this is a decoder for a DCF77 signal.
the decoder decodes the DCF77 signal and checks for a valid Date_Time.
since the dcf77 signal is only secured with a simple parity the decoder waits for two consecutive valid transmissions before it sets the output signals.
given a valid reception by the receiver the decoder can take up to 3 minutes to start its clocks the first time.
after a valid signal is detected the error output goes low and dignals a valid dcf signal from the receiver.
a tp is only valid for one program cycle to allow for external rtc setting.
after a valid signal is detected two independent internal clocks are started (RTC and RTC1), the seconds  of these clocks are generated by software since the dcf signal is only valid for minutes.
rtc is always utc ( world time) and rtc1 can be set to any time zone by setting the time_zone_offset and enabling dst for automatic summertime.
a sync output signals the the rtc and rtc1 are in sync with the dcf77 signal, if the dcf77 signal is lost for more then the sync time the sync output goes low
but the rtc and rtc1 outputs keep running based on software timing until a valid dcf77 signal is received again and triggers the clock.
in addition a millisecond output gives further resolutionof the clocks.
a dst output shows if daylight saving time is enables and the weekday output shows which day of week currently is ( 1= monday ... 7= sunday).

*)

(* if tp was set it should only be active for 1 cycle *)
TP := FALSE;

(* read system time *)
t1 := DWORD_TO_TIME(T_PLC_MS());
tx := t1 - last;

IF rec XOR edge THEN
	edge := rec;
	IF NOT rec AND tx > t#1700ms AND tx < t#2000ms THEN
		(* start condition reached *)
		state := 0;
		tp := NOT error;
	ELSIF NOT rec AND tx > t#700ms AND tx < t#1000ms THEN
		(* second switch detected *)
		IF state < 58 THEN state := state +1; ELSE state := 0; END_IF;
	ELSIF rec AND tx  < t#120ms THEN
		(* bit 0 detected  *)
		bits[state] := 0;
	ELSIF rec AND tx > t#120ms AND tx < t#250ms THEN
		(* bit 1 detected *)
		bits[state] := 1;
	ELSE
		(* error condition received signal is not valid *)
		error := TRUE;
		state := 0;
	END_IF;
	last := last + tx;
	IF rec AND state = 58 THEN
		error := FALSE;

		(* decode the bits and check for possible errors *)
		IF bits[0] OR NOT (bits[17] XOR bits[18]) OR NOT bits[20] THEN error := TRUE; END_IF;
		(* decode minute *)
		MINUTE := 0;
		MINUTE.0 := bits[21];
		MINUTE.1 := bits[22];
		MINUTE.2 := bits[23];
		MINUTE.3 := bits[24];
		IF bits[25] THEN MINUTE := MINUTE + 10; END_IF;
		IF bits[26] THEN MINUTE := MINUTE + 20; END_IF;
		IF bits[27] THEN MINUTE := MINUTE + 40; END_IF;
		IF MINUTE > 59 OR (bits[21] XOR bits[22] XOR bits[23] XOR bits[24] XOR bits[25] XOR bits[26] XOR bits[27] XOR bits[28]) THEN error := TRUE; END_IF;

		(* decode hour *)
		HOUR := 0;
		HOUR.0 := bits[29];
		HOUR.1 := bits[30];
		HOUR.2 := bits[31];
		HOUR.3 := bits[32];
		IF bits[33] THEN HOUR := HOUR + 10; END_IF;
		IF bits[34] THEN HOUR := HOUR +20; END_IF;
		IF HOUR > 23 OR (bits[29] XOR bits[30] XOR bits[31] XOR bits[32] XOR bits[33] XOR bits[34] XOR bits[35]) THEN error := TRUE; END_IF;

		(* decode day of month *)
		day := 0;
		day.0 := bits[36];
		day.1 := bits[37];
		day.2 := bits[38];
		day.3 := bits[39];
		IF bits[40] THEN day := day + 10; END_IF;
		IF bits[41] THEN day := day + 20; END_IF;
		IF day > 31 THEN error := TRUE; END_IF;

		(* decode day of week *)
		wday := 0;
		wday.0 := bits[42];
		wday.1 := bits[43];
		wday.2 := bits[44];
		IF wday > 7 OR wday < 1 THEN error := TRUE; END_IF;

		(* decode month *)
		MONTH := 0;
		MONTH.0 := bits[45];
		MONTH.1 := bits[46];
		MONTH.2 := bits[47];
		MONTH.3 := bits[48];
		IF bits[49] THEN MONTH := MONTH +10; END_IF;
		IF MONTH > 12 THEN error := TRUE; END_IF;

		(* decode year *)
		YEAR := 0;
		YEAR.0 := bits[50];
		YEAR.1 := bits[51];
		YEAR.2 := bits[52];
		YEAR.3 := bits[53];
		IF bits[54] THEN YEAR := YEAR + 10; END_IF;
		IF bits[55] THEN YEAR := YEAR + 20; END_IF;
		IF bits[56] THEN YEAR := YEAR + 40; END_IF;
		IF bits[57] THEN YEAR := YEAR + 80; END_IF;

		(* check parity for bits 36 to 58 *)
		cnt := 0;
		FOR i := 36 TO 58 DO IF bits[i] THEN cnt := cnt + 1; END_IF; END_FOR;
		IF NOT EVEN(cnt) THEN error := TRUE; END_IF;

		(* time must be valid for two cycles to clear error flag *)
		IF NOT error THEN
			(* set outputs *)
			old_time := mez;
			IF YEAR >= 70 THEN YEAR := YEAR + 1900; ELSE YEAR := YEAR + 2000; END_IF;
			mez := SET_DT(YEAR,MONTH,day,HOUR,MINUTE,0);
			DS := bits[17];
			IF DS THEN
				UTC := DWORD_TO_DT(DT_TO_DWORD(mez) - 7200);
			ELSE
				UTC := DWORD_TO_DT(DT_TO_DWORD(mez) - 3600);
			END_IF;

			(* set trigger signal only if the receiver has received 2 successive minutes *)
			IF mez <> old_time + t#1m THEN error := TRUE ; END_IF;
		END_IF;
	END_IF;
END_IF;

(* this portion implements a free running clock which is triggered by the dcf77 signal *)
tz := DWORD_TO_TIME(INT_TO_DWORD(ABS(time_offset))* 3600000);

(* input sdt is copied to utc at first power up *)
IF NOT init OR SET THEN
	init := TRUE;
	utc := sdt;
	tp := TRUE;
	DS := DSI;
END_IF;

IF tp THEN
	rtc := utc;
	IF DS AND dst_en THEN
		IF time_offset < 0 THEN	rtc1 := rtc - tz + t#1h; ELSE rtc1 := rtc + tz + t#1h; END_IF;
	ELSE
		IF time_offset < 0 THEN rtc1 := rtc - tz; ELSE rtc1 := rtc + tz; END_IF;
	END_IF;
	sync := TRUE;
	last_sync := last;
	ty := last;
ELSIF rtc > DWORD_TO_DT(0) AND T1 - ty >= t#1s THEN
	rtc := rtc + t#1s;
	rtc1 := rtc1 + t#1s;
	ty := ty + t#1s;
	sync := ty - last_sync < sync_timeout AND last_sync > DWORD_TO_TIME(0);
	wday := DAY_OF_WEEK(DT_TO_DATE(rtc1));
	DS := dst_en AND DST(utc);
END_IF;
msec := TIME_TO_INT(t1 - ty);



(* decode information
bits		content
0			Bitwert immer 0
1 bis 14	reserviert für Betriebsinformationen (nicht für DCF77-Nutzer bestimmt)
15			Rufbit für Alarmierung der PTB-Mitarbeiter
			(bis Mai 2003: Bitwert = 0 falls normale Antenne in Verwendung; 1 = Backupantenne)
16			Bitwert = 1 falls ein Wechsel von MEZ nach MESZ oder umgekehrt bevorsteht; Dauer der Anzeige: 1 Stunde
17 + 18	gültige Zeit = MEZ, falls Bit 17=0 und Bit 18=1
			gültige Zeit = MESZ, falls Bit 17=1 und Bit 18=0
19			Bitwert = 1 falls innerhalb den nächsten 59 Minuten eine Schaltsekunde angeordnet ist. Beim Einfügen einer Schaltsekunde wird anstelle der 59. die 60. Sekundenmarke weggelassen und in der 58. erfolgt ausnahmsweise ein Trägerabfall.
20			Startbit für Zeitinformation (immer 1)
21 - 27		1, 2, 4, 8, 10, 20, 40 Minuten (bitweise Addition)
28			Prüfbit (gerade Parität) für die Bits 21-27
29 - 34		1, 2, 4, 8, 10, 20 Stunden (bitweise Addition)
35			Prüfbit (gerade Parität) für die Bits 29-34
36 - 41		Tagesnummer im aktuellen Monat: 1, 2, 4, 8, 10, 20 (bitweise Addition)
42 - 44		Tagesnummer in der aktuellen Woche: 1, 2, 4 (bitweise Addition)
45 - 49		Monatsnummer: 1, 2, 4, 8, 10 (bitweise Addition)
50 - 57		Jahr (zweistellig): 1, 2, 4, 8, 10, 20, 40, 80 (bitweise Addition)
58			Prüfbit (gerade Parität) füR die Bits 36-57

*)
(* revision history

hm 2.feb 2007		rev 1.1
	change wday and dst outputs when there is no dcf reception

hm	26.feb 2007		rev 1.2
	changed statements where t#1h would be substracted from DT.
	under certain conditions the compiler would crash translating this statement

hm	17. sep 2007	rev 1.3
	replaced time() with T_PLC_MS() for compatibility reasons

hm	24. oct 2007		rev 1.4
	changed dst calculation because function dst was upgraded no error in DCF77 only a change in DST

hm	12. nov 2007		rev 1.5
	changed time_offset from time to integer to allow for negative offset time zones

hm	8. dec 2007		rev 1.6
	corrected an error in time_zone calculation

hm 23. jan 2008		rev 1.7
	added sdt input which is used to initialize rtc and rtc1 during first cycle.

hm 16. mar 2008		rev 1.8
	changed output weekday to wday and dst to ds for compatibility reasons

hm	19. apr. 2008	rev 1.9
	added input dsi to allow to set daylight savings time when SDT is TRUE.
	added asynchronous SET input

hm	7. oct. 2008	rev 1.10
	changed function weekday to day_of_week

*)

END_FUNCTION_BLOCK

// POUs/Logic/gate logic/PARITY
FUNCTION PARITY : BOOL
VAR_INPUT
	in : DWORD;
END_VAR


(*
	version 1.3	18 feb 2008
	programmer 	hugo
	tested BY		hans

this function calculates the even parity of an input Dword
the output will be true if the amount of high bits are an odd number.

*)

WHILE in > 0 DO
	PARITY := PARITY XOR in.0 XOR in.1 XOR in.2 XOR in.3;
	in := SHR(in,4);
END_WHILE;

(* code before rev 1.2
WHILE in > 0 DO
	IF in.0 THEN cnt := cnt +1; END_IF;
	in := SHR(in,1);
END_WHILE;
IF (cnt MOD 2) = 1 THEN parity := TRUE; ELSE parity := FALSE; END_IF;
*)

(* revision history

rev 1.0 hm 1 sep 2006
	original version

rev 1.1 hm 10.9.2007
	changed algorithm to improve performance

rev 1.2	hm	8 dec 2007
	changed algorithm to improve performance

rev 1.3	hm	18 feb 2008
	changed algorithm to improve performance
*)

END_FUNCTION

// POUs/Engineering/control/DEAD_BAND
FUNCTION DEAD_BAND : REAL
VAR_INPUT
	X : REAL;
	L : REAL;
END_VAR


(*
version 1.2	18. jan. 2011
programmer 	hugo
tested by		oscat

DEAD_BAND ist eine lineare Übertragungsfunktion mit Totzone. Die Funktion verschiebt den positiven Teil der Kurve um +L und den negativen Teil der Kurve um -L.
DEAD_BAND = X - L wenn X > L)
DEAD_BAND = X + L wenn X < -L
DEAD_BAND = 0 wenn Abs(X) <= L

*)

IF X > L THEN
	DEAD_BAND := X - L;
ELSIF X < -L THEN
	DEAD_BAND := X + L;
ELSE
	DEAD_BAND := 0.0;
END_IF;


(* revision history
hm	2. nov. 2007	rev 1.0
	original version

hm	14. jun. 2008	rev 1.1
	improved performance

hm	18. jan. 2011	rev 1.2
	assign 0 before return
*)

END_FUNCTION

// POUs/Engineering/control/DEAD_BAND_A
FUNCTION_BLOCK DEAD_BAND_A
VAR_INPUT
	X : REAL;
	T : TIME;
	KL : REAL := 1.0;
	LM : REAL;
END_VAR
VAR_OUTPUT
	Y : REAL;
	L : REAL;
END_VAR
VAR
	tp1 : FT_PT1;
	tp2 : FT_PT1;
END_VAR


(*
version 1.1	11. mar. 2009
programmer 	hugo
tested by		oscat

DEAD_BAND ist eine lineare Übertragungsfunktion mit Totzone. Die Funktion verschiebt den positiven Teil der Kurve um -L und den negativen Teil der Kurve um +L.
DEAD_BAND = X wenn Abs(X) > L wenn Abs(X) > L
DEAD_BAND = 0 wenn Abs(X) <= L
Die Breite der Totzone wird automatisch aus dem Signalrauschen errechnet.

*)

(* filter the input signal *)
tp1(in := X, T:= T);

(* filter the HF portion to generate a stable L *)
tp2(in := ABS(tp1.out - X), T := MULTIME(T, 4.0));

(* now we determine L which is half the width of the dead band *)
L := MIN(KL * tp2.out, LM);

IF X > L THEN
	Y := X - L;
ELSIF X < -L THEN
	Y := X + L;
ELSE
	Y := 0.0;
END_IF;


(* revision history
hm	14. jun. 2008	rev 1.0
	original version

hm	11. mar. 2009	rev 1.1
	real constants updated to new systax using dot

*)

END_FUNCTION_BLOCK

// POUs/Time&Date/MULTIME
FUNCTION MULTIME : TIME
VAR_INPUT
	t : TIME;
	M : REAL;
END_VAR


(*
version 1.1	14 mar 2008
programmer 	hugo
tested by		tobias

multiplies a time by a real number and returns a time
*)

MULTIME := DWORD_TO_TIME(REAL_TO_DWORD(DWORD_TO_REAL(TIME_TO_DWORD(t))*M));

(* revision history
hm		2. oct 2006	rev 1.0
	original version

hm		14. mar 2008	rev 1.1
	rounded the result after the last digit

*)

END_FUNCTION

// POUs/Engineering/control/FT_PT1
FUNCTION_BLOCK FT_PT1
VAR_INPUT
	in : REAL;
	T : TIME;
	K : REAL := 1.0;
END_VAR
VAR_OUTPUT
	out : REAL;
END_VAR
VAR
	last : DWORD;
	tx: DWORD;
	init: BOOL;
END_VAR

(*
version 1.11	18. jan. 2011
programmer 	hugo
tested by		oscat

FT_PT1 is an low pass filter with a programmable time T and faktor K.
 
*)

(* read system time *)
tx := T_PLC_US();

(* startup initialisation *)
IF NOT init OR T = t#0s THEN
	init := TRUE;
	out := K * in;
ELSE
	out := out + (in * K - out) * DWORD_TO_REAL(Tx - last) / TIME_TO_REAL(T) * 1.0E-3;
	IF ABS(out) < 1.0E-20 THEN out := 0.0; END_IF;
END_IF;
last := tx;


(*
hm 1.1.2007	rev 1.1
	corrected error while startup value was not correct
	for very small time values real output would run out of range.

hm 3.1.2007	rev 1.2
	corrected an error for falling edge failures.
	added output faktor K.

hm 27. 2. 2007	rev 1.3
	output will be input during init for definitive startup condition.

hm	15.9.2007	rev 1.4
	changed time() to T_PLC_US() for compatibilitxy resons
	increased internal accuracy to Microseconds instead of Milliseconds

hm	23. oct 2007	rev 1.5
	added out := in to the init statements

hm	30. nov 2007	rev 1.6
	changed out to be K * in during initialization

hm	5. jan 2008	rev 1.7
	improved code for better performance

hm	16. mar. 2008	rev 1.8
	added type conversion to avoid warning under codesys 3.0

hm	14. jun. 2008	rev 1.9
	improved code

hm	11. mar. 2009	rev 1.10
	real constants updated to new systax using dot

hm	18. jan. 2011	rev 1.11
	avoid underrun of out
*)

END_FUNCTION_BLOCK

// POUs/Logic/gate logic/DEC_2
FUNCTION_BLOCK DEC_2
VAR_INPUT
	D: BOOL;
	A: BOOL;
END_VAR
VAR_OUTPUT
	Q0: BOOL;
	Q1: BOOL;
END_VAR


(*
version 1.1	3 Mar 2007
programmer 	hugo
tested by		tobias

a bit input will be decoded to the two outputs Q0 or Q1
dependent on the value of A
A=0 decodes to Q0 and A=1 decodes to Q1

*)

Q0 := D AND NOT A;
Q1 := D AND A;

(* revision history
hm 3.3.2007	rev 1.1
	rewritten in ST for better compatibility

*)

END_FUNCTION_BLOCK

// POUs/Logic/gate logic/DEC_4
FUNCTION_BLOCK DEC_4
VAR_INPUT
	D: BOOL;
	A0: BOOL;
	A1: BOOL;
END_VAR
VAR_OUTPUT
	Q0: BOOL;
	Q1: BOOL;
	Q2: BOOL;
	Q3: BOOL;
END_VAR


(*
version 1.1	3 Mar 2007
programmer 	hugo
tested by		tobias

a bit input will be decoded to one of the 4 outputs
dependent on the Adress on A0 and A1

executioin TIME on wago 750-841 = 9us
*)

Q0 := D AND NOT A0 AND NOT A1;
Q1 := D AND A0 AND NOT A1;
Q2 := D AND NOT A0 AND A1;
Q3 := D AND A0 AND A1;

(* revision history
hm 3.3.2007	rev 1.1
	rewritten in ST for better compatibility

*)

END_FUNCTION_BLOCK

// POUs/Logic/gate logic/DEC_8
FUNCTION_BLOCK DEC_8
VAR_INPUT
	D: BOOL;
	A0: BOOL;
	A1: BOOL;
	A2: BOOL;
END_VAR
VAR_OUTPUT
	Q0: BOOL;
	Q1: BOOL;
	Q2: BOOL;
	Q3: BOOL;
	Q4: BOOL;
	Q5: BOOL;
	Q6: BOOL;
	Q7: BOOL;
END_VAR
VAR
	X : INT;
END_VAR

(*
version 1.3	28. mar. 2009
programmer 	hugo
tested by		oscat

a bit input will be decoded to one of the 8 outputs
dependent on the Adress on A0, A1 and A2


*)

X.0 := A0; X.1 := A1; X.2 := A2;

Q0 := FALSE;
Q1 := FALSE;
Q2 := FALSE;
Q3 := FALSE;
Q4 := FALSE;
Q5 := FALSE;
Q6 := FALSE;
Q7 := FALSE;

CASE X OF
	0 : Q0 := D;
	1 : Q1 := D;
	2 : Q2 := D;
	3 : Q3 := D;
	4 : Q4 := D;
	5 : Q5 := D;
	6 : Q6 := D;
	7 : Q7 := D;
END_CASE;



(* revision history
hm 3. mar. 2007	rev 1.1
	rewritten in ST for better compatibility

hm	26. oct. 2008	rev 1.2
	code optimized

hm	28. mar. 2009	rev 1.3
	replaced multiple assignments
*)

END_FUNCTION_BLOCK

// POUs/String/DEC_TO_BYTE
FUNCTION DEC_TO_BYTE : BYTE
VAR_INPUT
	DEC : STRING(10);
END_VAR
VAR
	pt : POINTER TO BYTE;
	i: INT;
	X: BYTE;
	stop: INT;
END_VAR

(*
version 1.1	30. sep 2008
programmer 	hugo
tested by		oscat

DEC_TO_byte converts a decimal string into a byte.

*)

pt := ADR(dec);
stop := LEN(DEC);
FOR I := 1 TO stop DO
	(* read the first character and subtract 48 to get value in decimal 0 = 48 *)
	x := pt^;
	(* calculate the value of the digit *)
	IF X > 47 AND x < 58 THEN
		DEC_TO_BYTE := DEC_TO_BYTE * 10 + X - 48;
	END_IF;
	pt := pt + 1;
END_FOR;



(* revision histroy
hm	20. jun. 2008	rev 1.0
	original release

hm	30. sep.2008	rev 1.1
	changed length of input string from 20 to 10
	corrected an error where decoding of characters 8 and 9 would fail

*)

END_FUNCTION

// POUs/String/DEC_TO_DWORD
FUNCTION DEC_TO_DWORD : DWORD
VAR_INPUT
	DEC : STRING(20);
END_VAR
VAR
	pt : POINTER TO BYTE;
	i: INT;
	X: BYTE;
	stop: INT;
END_VAR

(*
version 1.1	30. sep. 2008
programmer 	hugo
tested by		oscat

DEC_TO_DWORD converts a decimal string into a DWORD.

*)

pt := ADR(dec);
stop := LEN(dec);
FOR I := 1 TO stop DO
	(* read the first character and subtract 48 to get value in decimal 0 = 48 *)
	x := pt^;
	(* calculate the value of the digit *)
	IF X > 47 AND x < 58 THEN
		DEC_TO_DWORD := DEC_TO_DWORD * 10 + X - 48;
	END_IF;
	pt := pt + 1;
END_FOR;



(* revision histroy
hm	20. jun. 2008	rev 1.0
	original release

hm	30. sep. 2008	rev 1.1
	corrected an error where decoding of characters 8 and 9 would fail
*)

END_FUNCTION

// POUs/String/DEC_TO_INT
FUNCTION DEC_TO_INT : INT
VAR_INPUT
	DEC : STRING(10);
END_VAR
VAR
	pt : POINTER TO BYTE;
	i: INT;
	X: BYTE;
	sign: BOOL;
	stop: INT;
END_VAR

(*
version 1.1	30. sep. 2008
programmer 	hugo
tested by	oscat

DEC_TO_INT converts a decimal string into an Integer.

*)

pt := ADR(dec);
stop := LEN(dec);
FOR I := 1 TO stop DO
	(* read the first character and subtract 48 to get value in decimal 0 = 48 *)
	x := pt^;
	(* calculate the value of the digit *)
	IF X > 47 AND x < 58 THEN
		DEC_TO_INT := DEC_TO_INT * 10 + X - 48;
	ELSIF X = 45 AND DEC_TO_INT = 0 THEN
		sign := TRUE;
	END_IF;
	pt := pt + 1;
END_FOR;
IF sign THEN DEC_TO_INT := -DEC_TO_INT; END_IF;


(* revision histroy
hm	20. jun. 2008	rev 1.0
	original release

hm	30. sep. 2008	rev 1.1
	changed length of input string from 20 to 10
	corrected an error where decoding of characters 8 and 9 would fail
*)

END_FUNCTION

// POUs/Mathematical/DEC1
FUNCTION DEC1 : INT
VAR_INPUT
	X : INT;
	N : INT;
END_VAR


(*
version 1.1	27. oct. 2008
programmer 	hugo
tested by	oscat

This is a decrement function which decrements the variable X by 1 and if 0 is reached, it begins with N-1 again.
_dec1(X,3) will generate 2,1,0,2,...

*)

IF X = 0 THEN
	DEC1 := N - 1;
ELSE
	DEC1 := X - 1;
END_IF;


(* this is a very elegant version but 50% slower
X := (X - 1 + N) MOD N;
*)


(* revision history
hm	13. oct. 2008	rev 1.0
	original version

hm	27. oct. 2008	rev 1.1
	added statement to return value for compatibility reasons

*)

END_FUNCTION

// POUs/Engineering/conversion/DEG_TO_DIR
FUNCTION DEG_TO_DIR : STRING(3)
VAR_INPUT
	DEG : INT;
	N : INT;
	L : INT;
END_VAR
VAR
	ly: INT;
END_VAR


(*
version 1.1	22. oct. 2008
programmer 	hugo
tested by		oscat

this function converts degrees in compass direction.
the function supports output in english (L=0) and german (L=1).

*)

IF L = 0 THEN ly := LANGUAGE.DEFAULT; ELSE ly := MIN(L, LANGUAGE.LMAX); END_IF;
DEG_TO_DIR := LANGUAGE.DIRS[ly, ((SHL(DEG,N-1) + 45) / 90) MOD SHL(INT#2,N)*SHR(INT#8,N)];



(*
DIR := ((SHL(DEG,N-1) + 45) / 90) MOD SHL(INT#2,N);
explanation :
DIR is calculated BY the following formula:
DIR := ((DIR + 45) / 90) MOD 4 if N = 1 digit
North = 0, East = 1 ....
DIR := ((DIR + 22,5) / 45) MOD 8 if N = 2 digit
convert to integer calculation
DIR := ((DIR*2 + 45) / 90) MOD 8
N = 0, NE = 1 ....
ther above formula replaces 2^N with shift for performance
*)



(* revision histroy
hm	11. jun. 2008	rev 1.0
	original release

hm	22. oct. 2008	rev 1.1
	changed size of string variables to 30
*)

END_FUNCTION

// POUs/String/DEL_CHARS
FUNCTION DEL_CHARS : STRING(STRING_LENGTH)
VAR_INPUT
	IN : STRING(STRING_LENGTH);
	CX : STRING(80);
END_VAR
VAR
	pos: INT := 1;
	stop: INT;
END_VAR


(*
version 1.0	18. jun. 2008
programmer 	hugo
tested by	oscat

del_chars deletes all characters from a string which are specified in CX.

*)

(* copy input string *)
DEL_CHARS := IN;
stop := LEN(in);
WHILE pos <= stop DO
	IF FIND(cx, MID(DEL_CHARS, 1, pos)) > 0 THEN
		(* wrong chracter needs to be deleted *)
		DEL_CHARS := DELETE(DEL_CHARS, 1, pos);
		stop := stop - 1;	(* the string is one character shorter now *)
	ELSE
		(* charcter not found skip to next one *)
		pos := pos + 1;
	END_IF;
END_WHILE;



(* revision history

hm		18. jun. 2008	rev 1.0		
	original version 


*)

END_FUNCTION

// POUs/Engineering/signal processing/DELAY_4
FUNCTION_BLOCK DELAY_4
VAR_INPUT
	in : REAL;
END_VAR
VAR_OUTPUT
	out1 : REAL;
	out2 : REAL;
	out3 : REAL;
	out4 : REAL;
END_VAR
VAR
	temp: REAL;
END_VAR

(*
version 1.1	19 jan 2007
programmer 	hugo
tested by		tobias

this function block delays input values by each programm cycle
after 4 cycles the in value has shifted to the out 4 and will be discarded after the next cycle
the blocks can be cascaded.

*)

out4 := out3;
out3 := out2;
out2 := out1;
out1 := temp;
temp := in;

(* revision history

hm 19.1.2007	rev 1.1
	added variable temp to add 1 delay  for q1

*)

END_FUNCTION_BLOCK

// POUs/Building/HLK/DEW_RH
FUNCTION DEW_RH : REAL
VAR_INPUT
	VC : REAL;
	T : REAL;
END_VAR

(*
version 1.2	13. mar. 2009
programmer 	hugo
tested by		tobias

this function calculates the relative humidity in air for a given temperature in °C and vapor concentration in Kg/m³..

*)

DEW_RH := LIMIT(0.0, VC / DEW_CON(1.0, T), 100.0);

(* code before rev 1.1
dew_rh := VC / dew_con(100,T) * 100;
IF dew_rh > 100 THEN dew_rh := 100; END_IF;
*)

(* revision history
hm	29. apr 2007	rev 1.0
	original version

hm	2. 12. 2007	rev 1.1
	new code for better performance

hm	13. mar. 2009	rev 1.2
	real constants updated to new systax using dot

*)

END_FUNCTION

// POUs/Building/HLK/DEW_TEMP
FUNCTION DEW_TEMP : REAL
VAR_INPUT
	RH : REAL;
	T : REAL;
END_VAR
VAR CONSTANT
	a : REAL := 7.5;
	b : REAL := 237.3;
END_VAR
VAR
	V : REAL;
END_VAR

(*
version 1.6	13. mar. 2009
programmer 	hugo
tested by		oscat

this function calculates the dew point for air given the temperature and relative humidity.
dew_temp(60,0.25) = 16.7 °C.
which means the dew point for air with 25° and 60% RH is at 16.7 °C.


*)

IF rh > 0.0 THEN
(*	old code was rewritten for better performance
	SDD := 6.1078*EXPT(10,(a*T)/(b+T));
	DD := RH/100 * SDD;
	V := LOG(DD/6.1078);
	dew_temp := b*V/(a-v);
*)
	V := LOG(RH * 0.01 * EXP10((a*T) / (b+T)));
	DEW_TEMP := b*V / (a-V);
ELSE
	DEW_TEMP:= phys.T0;
END_IF;

(* revision history

hm		2.10.2006	rev 1.0
	original version created

hm		29.4.2007	rev 1.1
	checked for rh not to be 0 because log(0) is not defined

hm		13.9.2007	rev 1.2
	code rewritten for better performance

hm	2. dec 2007	rev 1.3
	changed code for better performance

hm	8. jan 2008	rev 1.4
	further improvement in performance

hm	18. oct. 2008	rev 1.5
	using phys constants	

hm	13. mar. 2009	rev 1.6
	real constants updated to new systax using dot
	function will now return -273.15 °C for RH = 0
*)

(*
Bezeichnungen:
r = relative Luftfeuchte
T = Temperatur in °C
TK = Temperatur in Kelvin (TK = T + 273.15)
TD = Taupunkttemperatur in °C
DD = Dampfdruck in hPa
SDD = Sättigungsdampfdruck in hPa

Parameter:
a = 7.5, b = 237.3 für T >= 0
a = 7.6, b = 240.7 für T < 0 über Wasser (Taupunkt)
a = 9.5, b = 265.5 für T < 0 über Eis (Frostpunkt)

R* = 8314.3 J/(kmol*K) (universelle Gaskonstante)
mw = 18.016 kg (Molekulargewicht des Wasserdampfes)
AF = absolute Feuchte in g Wasserdampf pro m3 Luft

Formeln:

   1. SDD(T) = 6.1078 * 10^((a*T)/(b+T))
   2. DD(r,T) = r/100 * SDD(T)
   3. r(T,TD) = 100 * SDD(TD) / SDD(T)
   4. TD(r,T) = b*v/(a-v) mit v(r,T) = log10(DD(r,T)/6.1078)
   5. AF(r,TK) = 10^5 * mw/R* * DD(r,T)/TK; AF(TD,TK) = 10^5 * mw/R* * SDD(TD)/TK 

*)

END_FUNCTION

// POUs/Building/electrical/DIMM_2
FUNCTION_BLOCK DIMM_2
VAR_INPUT
	SET : BOOL;
	VAL : BYTE := 255;
	I1 : BOOL;
	I2 : BOOL;
	RST : BOOL;
END_VAR
VAR_INPUT CONSTANT
	T_DEBOUNCE : TIME := T#10ms;
	T_ON_MAX : TIME := T#0h;
	T_DIMM_START : TIME := T#1s;
	T_DIMM: TIME := T#3s;
	MIN_ON : BYTE := 50;
	MAX_ON : BYTE := 255;
	RST_OUT : BOOL := TRUE;
	SOFT_DIMM : BOOL := TRUE;
	DBL1_TOG : BOOL;
	DBL2_TOG : BOOL;
	DBL1_SET : BOOL;
	DBL2_SET : BOOL;
	DBL1_POS : BYTE;
	DBL2_POS : BYTE;
END_VAR
VAR_OUTPUT
	Q : BOOL := FALSE;
	D1 : BOOL;
	D2 : BOOL;
END_VAR
VAR_IN_OUT
	OUT : BYTE;
END_VAR
VAR
	t1, t2 : TOF;
	dc1, dc2 : CLICK_MODE;
	t3 : TON;
	dim : _RMP_B;
END_VAR

(*
version 1.0	22. mar. 2009
programmer 	hugo
tested by	tobias

this is an intelligent dimmer interface with an autoset feature using double switch inputs
a configurable debounce timer will debounce the input signals
if t_on_max is set to anything other then 0 the output will be turned off after the max on time is reached.
the times for debounce, dimming ramp, wait time before dimming and max on time are all programmable.

the dimmer has outputs Q for on and off and also out with the analog dimm value.
two additional outputs d1 and d2 decode double clicks on i1 and i2.

*)

(* debouncing for inputs i1 and i2 *)
t1(IN := I1, PT := T_DEBOUNCE);
t2(IN := I2, PT := T_DEBOUNCE);
dc1(in := t1.Q, T_LONG := T_DIMM_START);
dc2(in := t2.Q, T_LONG := T_DIMM_START);


IF RST THEN
	IF RST_OUT THEN out := 0; END_IF;
	Q := FALSE;
	D1 := FALSE;
	D2 := FALSE;
ELSIF set THEN
	OUT := VAL;
	Q := TRUE;
ELSIF dc1.SINGLE THEN
	(* single click on i1 turns the dimmer on *)
	out := LIMIT(MAX(MIN_ON,1), out, MAX_ON);
	Q := TRUE;
ELSIF dc2.SINGLE THEN
	(* single click on i2 turns the dimmer off *)
	Q := FALSE;
ELSIF dc1.TP_LONG THEN
	(* continuous on at i1 dimms up *)
	IF NOT Q THEN
		out := SEL(SOFT_DIMM, LIMIT(MAX(MIN_ON,1), out, MAX_ON), 1);
	END_IF;
	Q := TRUE;
	dim.DIR := TRUE;
ELSIF dc2.TP_LONG THEN
	(* continuous on at i2 dimms down *)
	dim.DIR := FALSE;
END_IF;

(* set the double click output *)
IF NOT DBL1_TOG THEN D1 := FALSE; END_IF;
IF dc1.DOUBLE THEN
	IF DBL1_SET THEN
		OUT := DBL1_POS;
		Q := TRUE;
	ELSE
		D1 := NOT D1;
	END_IF;
END_IF;
IF NOT DBL2_TOG THEN D2 := FALSE; END_IF;
IF dc2.DOUBLE THEN
	IF DBL2_SET THEN
		OUT := DBL2_POS;
		Q := TRUE;
	ELSE
		D2 := NOT D2;
	END_IF;
END_IF;


(* while dimming is active ramp the output out up or down *)
dim(dir := dc2.LONG, e := dc1.LONG OR dc2.LONG , TR := T_DIMM, rmp := out);

(* turn off output if a value of 0 is reached *)
IF out = 0 THEN Q := FALSE; END_IF;

(* limit the maximum runtime *)
IF t_ON_MAX > t#0s THEN
	t3(in := q, pt := T_ON_MAX);
	Q := Q XOR t3.Q;
END_IF;




(* revision history

hm 22. mar. 2009	rev 1.0
	original version

*)

END_FUNCTION_BLOCK

// POUs/Building/electrical/DIMM_I
FUNCTION_BLOCK DIMM_I
VAR_INPUT
	SET : BOOL;
	VAL : BYTE := 255;
	IN : BOOL;
	RST : BOOL;
END_VAR
VAR_INPUT CONSTANT
	T_DEBOUNCE : TIME := T#10ms;
	T_RECONFIG : TIME := T#10s;
	T_ON_MAX : TIME := T#0h;
	T_DIMM_START : TIME := T#1s;
	T_DIMM: TIME := T#3s;
	MIN_ON : BYTE := 50;
	MAX_ON : BYTE := 255;
	SOFT_DIMM : BOOL := TRUE;
	DBL_toggle : BOOL;
	RST_OUT : BOOL;
END_VAR
VAR_OUTPUT
	Q : BOOL := FALSE;
	DBL : BOOL;
END_VAR
VAR_IN_OUT
	OUT : BYTE;
END_VAR
VAR
	config : SW_RECONFIG;
	decode : CLICK_MODE;
	t3 : TON;
	dim : _RMP_B;
	dir : BOOL;
END_VAR

(*
version 2.3	26. jan. 2009
programmer 	hugo
tested by		tobias

this is an intelligent dimmer interface with an autoset feature for "in" it will automatically detect the type of switch:
low active pulses or high high active pulses are allowd for in.
a configurable debounce timer will debounce input signals
if t_on_max is set to anything other then 0 the output will be turned off after the max on time is reached.
the times for debounce, dimming ramp, wait time before dimming and max on time are all programmable.

the dimmer has outputs Q for on and off and also out with the analog dimm value.

*)

(* the input is first sent through auto reconfiguration and debouncing *)
config(IN := IN, TD := T_DEBOUNCE, TR := T_RECONFIG);
decode(in := config.Q, T_LONG := T_DIMM_START);

IF RST THEN
	IF rst_out THEN out := 0; END_IF;
	Q := FALSE;
	dir := out > 127;
ELSIF set THEN
	out := val;
	Q := TRUE;
	(* set direction to up when value < 127 otherwise set dir down dir is reversed because next action will reverse again *)
	dir := out > 127;
ELSIF decode.SINGLE THEN
	(* a single click reverses output Q *)
	Q := NOT Q;
	(* when dimmer is turned on we need to limit out to min and max limits *)
	IF Q THEN	out := LIMIT(MAX(MIN_ON,1), out, MAX_ON);	END_IF;
	(* set the appropriate direction of dimmer dir is reversed because next action will reverse again *)
	dir := out > 127;
ELSIF decode.TP_LONG THEN
	IF NOT Q THEN
		IF SOFT_DIMM THEN
			OUT := 1;
			dir := TRUE;
		ELSE
			OUT := LIMIT(MAX(MIN_ON,1), out, MAX_ON);
			DIR := out < 127;
		END_IF;
		Q := TRUE;
	ELSE
		(* reverse direction with every long click *)
		dir := NOT dir;
	END_IF;
END_IF;

(* set the double click output *)
IF NOT dbl_toggle THEN dbl := FALSE; END_IF;
IF decode.DOUBLE THEN dbl := NOT dbl; END_IF;

(* while dimming is active ramp the output out up or down *)
dim(DIR := dir, e := decode.LONG AND Q, TR := T_DIMM, rmp := out);

(* reverse direction when limits are reached *)
IF out = 0 THEN
	dir := TRUE;
ELSIF out = 255 THEN
	dir := FALSE;
END_IF;

(* limit the maximum runtime *)
IF t_ON_MAX > t#0s THEN
	t3(in := q, pt := T_ON_MAX);
	Q := Q XOR t3.Q;
END_IF;




(* revision history

hm 22.1.2007		rev 1.1
	deleted unused structure ramp

hm 2.feb 2007		rev 1.2
	changed structure to read time() at the beginning for better time consistency if a higher priorized tak interrupts dimm_i
	added statements in case structure for state 1 to allow for short 1 cycle input pulses

hm 	15.9.2007		rev 1.3
	replaced Time() with T_PLC_MS for compatibility and performance reasons

hm	30. sep. 2008	rev 1.4
	added Input VAL to supply value for set input
	added setup parameter init_val

hm	22. oct. 2008	rev 2.0
	new code and features

hm	14. nov. 2008	rev 2.1
	added soft_dimm feature

hm	16. nov. 2008	rev 2.2
	added reset out feature

hm	26. jan. 2009	rev 2.3
	dimming will also reverse at out = 0
	rst will override set
*)

END_FUNCTION_BLOCK

// POUs/Engineering/conversion/DIR_TO_DEG
FUNCTION DIR_TO_DEG : INT
VAR_INPUT
	DIR : STRING(3);
	L : INT;
END_VAR
VAR
	ly: INT;
	i : INT;
END_VAR

(*
version 1.1	22. oct. 2008
programmer 	hugo
tested by	oscat

this function converts compass directions to degrees
it will recognize up to 3 letter directions in english and german writing.

*)

IF L = 0 THEN ly := LANGUAGE.DEFAULT; ELSE ly := MIN(L, LANGUAGE.LMAX); END_IF;
FOR i := 0 TO 15 DO
	IF language.DIRS[ly, i] = DIR THEN EXIT; END_IF;
END_FOR;
DIR_TO_DEG := SHR(i * 45 + 1, 1);






(* revision histroy
hm	22. oct. 2008	rev 1.1
	original release

*)

END_FUNCTION

// POUs/Engineering/automation/DRIVER_1
FUNCTION_BLOCK DRIVER_1
VAR_INPUT CONSTANT
	Toggle_Mode : BOOL;
	Timeout : TIME;
END_VAR
VAR_INPUT
	SET : BOOL;
	IN : BOOL;
	RST : BOOL;
END_VAR
VAR_OUTPUT
	Q : BOOL;
END_VAR
VAR
	off : TON;
	edge: BOOL;
END_VAR

(*
version 1.0	2 jan 2008
programmer 	hugo
tested by		tobias

driver_1 is a multi purpose driver.
a rising edge on in sets the output high if toggle is flase. while toggle is true, a rising edge on in toggles the output Q.
if a timeout is specified the output q will be reset to false automatically after the timeout has elapsed.
a asynchronous reset and set will force the output high or low respectively.

*)

IF off.Q THEN Q := FALSE; END_IF;
IF rst THEN
	Q := FALSE;
ELSIF set THEN
	Q := TRUE;
ELSIF IN AND NOT edge THEN
	IF toggle_mode THEN q := NOT Q; ELSE q := TRUE; END_IF;
END_IF;
edge := in;
IF timeout > t#0s THEN off(in := Q, PT := Timeout); END_IF;


(* revision history
hm	2. jan 2008		rev 1.0
	original version

*)

END_FUNCTION_BLOCK

// POUs/Engineering/automation/DRIVER_4
FUNCTION_BLOCK DRIVER_4
VAR_INPUT CONSTANT
	Toggle_Mode : BOOL;
	Timeout : TIME;
END_VAR
VAR_INPUT
	SET : BOOL;
	IN0, IN1, IN2, IN3 : BOOL;
	RST : BOOL;
END_VAR
VAR_OUTPUT
	Q0, Q1, Q2, Q3 : BOOL;
END_VAR
VAR
	d0, d1, d2, d3 : DRIVER_1;
END_VAR

(*
version 1.0	2 jan 2008
programmer 	hugo
tested by		tobias

driver_4 is a 4 channel multi purpose driver.
a rising edge on in? sets the output Q? high if toggle_mode is flase. while toggle_mode is true, a rising edge on in? toggles the output Q?.
if a timeout is specified the output Q? will be reset to false automatically after the timeout has elapsed.
a asynchronous reset and set will force the output high or low respectively.
an asynchronous set will force all outputs high simultaneously

*)

D0(Set:=set, in:=in0, rst:=rst, toggle_mode:=toggle_mode, timeout:=timeout);
D1(Set:=set, in:=in1, rst:=rst, toggle_mode:=toggle_mode, timeout:=timeout);
D2(Set:=set, in:=in2, rst:=rst, toggle_mode:=toggle_mode, timeout:=timeout);
D3(Set:=set, in:=in3, rst:=rst, toggle_mode:=toggle_mode, timeout:=timeout);
Q0 := D0.Q;
Q1 := D1.Q;
Q2 := D2.Q;
Q3 := D3.Q;


(* revision history
hm	2. jan 2008		rev 1.0
	original version

*)

END_FUNCTION_BLOCK

// POUs/Engineering/automation/DRIVER_4C
FUNCTION_BLOCK DRIVER_4C
VAR_INPUT
	IN : BOOL;
	RST : BOOL;
END_VAR
VAR_INPUT CONSTANT
	Timeout : TIME;
	SX : ARRAY[1..7] OF BYTE :=[ 1,3,7,15];
END_VAR
VAR_OUTPUT
	SN : INT;
	Q0 : BOOL;
	Q1 : BOOL;
	Q2 : BOOL;
	Q3 : BOOL;
END_VAR
VAR
	off : TON;
	edge: BOOL;
END_VAR

(*
version 1.0	23. mar. 2009
programmer 	hugo
tested by	tobias

driver_4C is a multi purpose driver.
a rising edge on in switches from S0 state S1 and the next edge to state S2 and so on.
in state S0 all outputs Q are FALSE.
The stet of the Outputs in any state S? is configurable with setup variables.
The variables S1..S5 define the states, while the sequence is terminated when a state Variable S? = 0.
The lower bits 0..3 of the state vars S? are corresponding to the Outputs Q0..Q3

*)

IF RST OR off.Q THEN
	SN := 0;
ELSIF IN AND NOT edge THEN
	SN := SN + 1;
	IF SN > 7 OR SX[SN] = 0 THEN SN := 0; END_IF;
END_IF;
edge := in;
IF SN > 0 THEN
	Q0 := SX[SN].0;
	Q1 := SX[SN].1;
	Q2 := SX[SN].2;
	Q3 := SX[SN].3;
ELSE
	Q0 := FALSE;
	Q1 := FALSE;
	Q2 := FALSE;
	Q3 := FALSE;
END_IF;

(* maximaum timeout *)
IF timeout > t#0s THEN off(in := SN > 0, PT := Timeout); END_IF;


(* revision history
hm	23. mar. 2009	rev 1.0
	original version

*)

END_FUNCTION_BLOCK

// POUs/Engineering/measurements/DT_SIMU
FUNCTION_BLOCK DT_SIMU
VAR_INPUT
	START : DT;
	SPEED : REAL := 1.0;
END_VAR
VAR_OUTPUT
	DTS : DT;
END_VAR
VAR
	tc : DWORD;
	init: BOOL;
	last: DWORD;
	tx: DWORD;
	td: DWORD;
END_VAR

(*
version 1.2	8. mar. 2009
programmer 	hugo
tested by		oscat

DT_SIMU simulates a real time clock and can be adjusted to different speeds
it can also be used in simulation to simulate a real time clock.
the peed of the clock can be increased or decreased to debug timers.
with the input start a start date-time can be specified.

*)

(* read system timer *)
tx := T_PLC_MS();
tc := REAL_TO_DWORD(DWORD_TO_REAL(tx - last) * speed);

IF NOT init THEN
	init := TRUE;
	DTS := Start;
	tc := 0;
	last := tx;
ELSIF SPEED = 0.0 THEN
	DTS := DWORD_TO_DT(DT_TO_DWORD(DTS) + 1);
ELSIF tc >= 1000 THEN
	td := (tc / 1000) * 1000;
	DTS := DTS + DWORD_TO_TIME(td);
	last := last + REAL_TO_DWORD(DWORD_TO_REAL(td) / speed);
END_IF;

(* revision history
hm	11. sep. 2008	rev 1.0
	original version

hm	16. nov	2008	rev 1.1
	added type conversions for compatibility reasons

hm	8.	mar. 2009	rev 1.2
	added increment by cycle mode

*)

END_FUNCTION_BLOCK

// POUs/Time&Date/DT_TO_SDT
FUNCTION DT_TO_SDT : SDT
VAR_INPUT
	DTI : DT;
END_VAR
VAR
	tmp : DATE;
	tdt : DWORD;
END_VAR


(*
version 1.0	18. oct 2008
programmer 	hugo
tested by	oscat

converts date_time to Structured date time (SDT)

*)

tmp := DT_TO_DATE(dti);
tdt := DT_TO_DWORD(dti) - DATE_TO_DWORD(tmp);
DT_TO_SDT.YEAR := YEAR_OF_DATE(tmp);
DT_TO_SDT.MONTH := MONTH_OF_DATE(tmp);
DT_TO_SDT.DAY := DAY_OF_MONTH(tmp);
DT_TO_SDT.WEEKDAY := DAY_OF_WEEK(tmp);
DT_TO_SDT.SECOND := DWORD_TO_INT(tdt MOD 60);
DT_TO_SDT.MINUTE := DWORD_TO_INT((tdt / 60) MOD 60);
DT_TO_SDT.HOUR := DWORD_TO_INT(tdt / 3600);

(* revision history

hm 18. oct. 2008	rev 1.0
	original version

*)

END_FUNCTION

// POUs/String/DT_TO_STRF
FUNCTION DT_TO_STRF : STRING
VAR_INPUT
	DTI : DT;
	MS : INT;
	FMT : STRING;
	LANG : INT;
END_VAR
VAR CONSTANT
	FILL : STRING(1) := '0';
	BLANK : STRING(1) := ' ';
END_VAR
VAR
	ly : INT;
	dx: DATE;
	fs: STRING(10);
	td: TOD;
	tmp : INT;
	pos : INT;
	f : INT;
END_VAR

(*
version 1.1	19. oct. 2008
programmer 	hugo
tested by	oscat

DT_TO_STRINGF converts a DATETIME input to a formatted string

*)

IF LANG < 1 THEN ly := language.DEFAULT; ELSE ly := MIN(language.LMAX, LANG); END_IF;

(* decode date and time information *)
dx := DT_TO_DATE(DTI);
td := DT_TO_TOD(DTI);

(* parse the format string *)
DT_TO_STRF := FMT;
pos := FIND(DT_TO_STRF, '#');
WHILE pos > 0 DO
	(* retrieve format identifier *)
	f := CODE(DT_TO_STRF, pos + 1);
	(* generate the return string according to the format character *)
	fs := '';
	CASE f OF
		65 : (* letter A retunrs the year in 4 digits *)
			fs := INT_TO_STRING(YEAR_OF_DATE(dx));
		66 : (* letter B returns the year in exactly 2 digits *)
			fs := RIGHT(INT_TO_STRING(YEAR_OF_DATE(dx)),2);
		67 : (* letter C returns the month with 1 or 2 digits *)
			fs := INT_TO_STRING(MONTH_OF_DATE(dx));
		68 : (* letter D returns the month with exactly 2 digits *)
			fs := INT_TO_STRING(MONTH_OF_DATE(dx));
			IF LEN(fs) < 2 THEN fs := CONCAT('0', fs); END_IF;
		69 : (* letter E returns the month with 3 characters *)
			fs := MONTH_TO_STRING(MONTH_OF_DATE(dx), ly, 3);
		70 : (* letter F returns the month with all characters *)
			fs := MONTH_TO_STRING(MONTH_OF_DATE(dx), ly, 0);
		71 : (* letter G returns the day with up to 2 digits *)
			fs := INT_TO_STRING(DAY_OF_MONTH(dx));
		72 : (* letter H returns the day of the month with exactly 2 digits *)
			fs := INT_TO_STRING(DAY_OF_MONTH(dx));
			IF LEN(fs) < 2 THEN fs := CONCAT(FILL, fs); END_IF;
		73 : (* letter I returns the weekday as the number 1..7 1 = monday *)
			fs := INT_TO_STRING(DAY_OF_WEEK(dx));
		74 : (* letter J returns the weekday in 2 character writing *)
			fs := WEEKDAY_TO_STRING(DAY_OF_WEEK(dx), ly, 2);
		75 : (* letter K returns the weekday with all characters *)
			fs := WEEKDAY_TO_STRING(DAY_OF_WEEK(dx), ly, 0);
		76 : (* letter L returns AM or PM for the given DateTime *)
			IF td >= TOD#12:00 THEN fs := 'PM'; ELSE fs := 'AM'; END_IF;
		77 : (* letter M returns the hour in 1 or 2 digit form 0..24h *)
			fs := INT_TO_STRING(HOUR(td));
		78 : (* letter N returns the hour in exactly 2 digit form 0..24h *)
			fs := INT_TO_STRING(HOUR(td));
			IF LEN(fs) < 2 THEN fs := CONCAT(FILL, fs); END_IF;
		79 : (* letter O returns the hour in 1 or 2 digit form 0..12h *)
			tmp := HOUR(td) MOD 12;
			IF tmp = 0 THEN tmp := 12; END_IF;
			fs := INT_TO_STRING(tmp);
		80 : (* letter P returns the hour in exactly 2 digit form 0..12h *)
			tmp := HOUR(td) MOD 12;
			IF tmp = 0 THEN tmp := 12; END_IF;
			fs := INT_TO_STRING(tmp);
			IF LEN(fs) < 2 THEN fs := CONCAT(FILL, fs); END_IF;
		81 : (* letter Q returns the minute of the hour in 1 or two digit form *)
			fs := INT_TO_STRING(MINUTE(td));
		82 : (* letter R returns the minute of the hour in exactly two digit form *)
			fs := INT_TO_STRING(MINUTE(td));
			IF LEN(fs) < 2 THEN fs := CONCAT(FILL, fs); END_IF;
		83 : (* letter S returns the second of the minute in 1 or two digit form *)
			fs := INT_TO_STRING(REAL_TO_INT(SECOND(td)));
		84 : (* letter T returns the second of the minute in exactly two digit form *)
			fs := INT_TO_STRING(REAL_TO_INT(SECOND(td)));
			IF LEN(fs) < 2 THEN fs := CONCAT(FILL, fs); END_IF;
		85 : (* letter U returns the milliseconds in 1 to 3 digits *)
			fs := INT_TO_STRING(MS);
		86 : (* letter V returns the milliseconds in exactly 3 digit form *)
			fs := INT_TO_STRING(MS);
			fs := CONCAT('00',fs);
			fs := RIGHT(fs, 3);
		87 : (* letter W returns the day of the month with exactly 2 digits first digit is filled with blank if necessary *)
			fs := INT_TO_STRING(DAY_OF_MONTH(dx));
			IF LEN(fs) < 2 THEN fs := CONCAT(BLANK, fs); END_IF;
		88 : (* letter X returns the month with exactly 2 digits first digit is filled with blank if necessary *)
			fs := INT_TO_STRING(MONTH_OF_DATE(dx));
			IF LEN(fs) < 2 THEN fs := CONCAT(BLANK, fs); END_IF;
		END_CASE;
	DT_TO_STRF := REPLACE(DT_TO_STRF, fs, 2, pos);
	pos := FIND(DT_TO_STRF, '#');
END_WHILE;


(* revision history
hm	7. oct. 2008	rev 1.0
	original version

hm	19. oct. 2008	rev 1.1
	changed language setup constants
*)

END_FUNCTION

// POUs/String/MONTH_TO_STRING
FUNCTION MONTH_TO_STRING : STRING(10)
VAR_INPUT
	MTH : INT;
	LANG : INT;
	LX : INT;
END_VAR
VAR
	ly : INT;
END_VAR

(*
version 1.1	19. oct. 2008
programmer 	hugo
tested by	oscat

MONTH_TO_STRING converts an Integer 1..12 into a String with the Names of the corresponding Month.
the decoding is according to the language setup in global vars

*)

IF LANG = 0 THEN Ly := LANGUAGE.DEFAULT; ELSE ly := MIN(LANG, language.LMAX); END_IF;
IF MTH < 1 OR MTH > 12 THEN
	RETURN;
ELSIF LX = 0 THEN
	MONTH_TO_STRING := language.MONTHS[ly, MTH];
ELSIF Lx = 3 THEN
	MONTH_TO_STRING := language.MONTHS3[ly, MTH];
END_IF;


(* revisison history

hm	21. sep. 2008	rev 1.0
	original version

hm	19. oct. 2008	rev 1.1
	changed language setup constants
*)

END_FUNCTION

// POUs/String/WEEKDAY_TO_STRING
FUNCTION WEEKDAY_TO_STRING : STRING(10)
VAR_INPUT
	WDAY : INT;
	LANG : INT;
	LX : INT;
END_VAR
VAR
	ly : INT;
END_VAR

(*
version 1.1	19. oct. 2008
programmer 	hugo
tested by	oscat

WEEKDAY_TO_STRING converts an Integer 1..7 into a String with the Names of the corresponding weekday.
the decoding is according to the language setup in global vars

*)

IF LANG = 0 THEN ly := LANGUAGE.DEFAULT; ELSE ly := MIN(LANG, LANGUAGE.LMAX); END_IF;
IF wday < 1 OR wday > 7 THEN
	RETURN;
ELSIF LX = 0 THEN
	WEEKDAY_TO_STRING := language.WEEKDAYS[ly, WDAY];
ELSIF Lx = 2 THEN
	WEEKDAY_TO_STRING := language.WEEKDAYS2[ly, WDAY];
END_IF;


(* revisison history

hm	21. sep. 2008	rev 1.0
	original version

hm	19. oct. 2008	rev 1.1
	changed language setup constants
*)

END_FUNCTION

// POUs/Time&Date/DT2_TO_SDT
FUNCTION DT2_TO_SDT : SDT
VAR_INPUT
	DI : DATE;
	TI : TOD;
END_VAR


(*
version 1.0	18. oct 2008
programmer 	hugo
tested by	oscat

converts date and time of day to Structured date time (SDT)

*)

DT2_TO_SDT.YEAR := YEAR_OF_DATE(di);
DT2_TO_SDT.MONTH := MONTH_OF_DATE(di);
DT2_TO_SDT.DAY := DAY_OF_MONTH(di);
DT2_TO_SDT.WEEKDAY := DAY_OF_WEEK(di);
DT2_TO_SDT.MS := DWORD_TO_INT(TOD_TO_DWORD(ti) MOD 1000);
DT2_TO_SDT.SECOND := DWORD_TO_INT((TOD_TO_DWORD(ti) / 1000) MOD 60);
DT2_TO_SDT.MINUTE := DWORD_TO_INT((TOD_TO_DWORD(ti) / 60000) MOD 60);
DT2_TO_SDT.HOUR := DWORD_TO_INT(TOD_TO_DWORD(ti) / 3600000);

(* revision history

hm 18. oct. 2008	rev 1.0
	original version

*)

END_FUNCTION

// POUs/Logic/gate logic/DW_TO_REAL
FUNCTION DW_TO_REAL : REAL
VAR_INPUT
	X : DWORD;
END_VAR
VAR
	pt : POINTER TO REAL;
END_VAR

(*
version 1.0	18. apr. 2008
programmer 	hugo
tested by		tobias

this function converts a DWORD to REAL in a bitwise manner.
*)

pt := ADR(X);
DW_TO_REAL := pt^;

(* revision history
hm	18. apr. 2008
	original version

*)

END_FUNCTION

// POUs/Logic/gate logic/DWORD_OF_BYTE
FUNCTION DWORD_OF_BYTE : DWORD
VAR_INPUT
	B3 : BYTE;
	B2 : BYTE;
	B1 : BYTE;
	B0 : BYTE;
END_VAR


(*
version 1.3	18. jul. 2009
programmer 	hugo
tested by		tobias

this function creates a Dword from 4 individual bytes

*)

DWORD_OF_BYTE := SHL(SHL(SHL(BYTE_TO_DWORD(B3),8) OR BYTE_TO_DWORD(B2),8) OR BYTE_TO_DWORD(B1),8) OR BYTE_TO_DWORD(B0);


(* revision history
hm	24. jan 2007	rev 1.0
	original version

hm 2. jan 2008	rev 1.1
	inproved performance

hm	23. apr. 2008	rev 1.2
	reverse order of inputs to be more logical

hm	18. jul. 2009	rev 1.3
	added type conversions for compatibility reasons
*)

END_FUNCTION

// POUs/Logic/gate logic/DWORD_OF_WORD
FUNCTION DWORD_OF_WORD : DWORD
VAR_INPUT
	W1 : WORD;
	W0 : WORD;
END_VAR


(*
version 1.0	18. jul. 2009
programmer 	hugo
tested by		tobias

this function creates a Dword from 2 individual Words

*)

DWORD_OF_WORD := SHL(WORD_TO_DWORD(W1),16) OR WORD_TO_DWORD(W0);


(* revision history

hm	18. jul. 2009	rev 1.0
	original version

*)

END_FUNCTION

// POUs/String/DWORD_TO_STRB
FUNCTION DWORD_TO_STRB : STRING(32)
VAR_INPUT
	IN : DWORD;
END_VAR
VAR
	pt : POINTER TO BYTE;
	i: INT;
END_VAR

(*
version 1.3	20. jun. 2008
programmer 	hugo
tested by	oscat

DWORD_TO_STRINGB converts a DWORD to a String of Bits represented by '0' and '1' s.
The lowest order bit will be on the right and the high order bit on the left.

*)

(* pointer für die ausgabe ermitteln *)
pt := ADR(DWORD_TO_STRB);
(* die 8 ausgabecharacter ermitteln und schreiben *)
FOR i := 1 TO 32 DO
	pt^:= BOOL_TO_BYTE(in.31) + 48;
	in := SHL(in,1);
	pt := pt + 1;
END_FOR;

(* der ausgabestring muss nochg mit 0 abgeschlossen werden *)
pt^ := 0;

(* revision history
hm		9.6.2007	rev 1.0		
	original version

hm		15.dec 2007	rev 1.1
	changed code for better performance

hm	29. mar. 2008	rev 1.2
	changed STRING to STRING(32)

hm	20. jun. 2008	rev 1.3
	performance improvement

*)

END_FUNCTION

// POUs/String/DWORD_TO_STRF
FUNCTION DWORD_TO_STRF : STRING(20)
VAR_INPUT
	IN : DWORD;
	N : INT;
END_VAR


(*
version 1.0	26 jan 2007
programmer 	hugo
tested by		tobias

dword_to_strF converts a DWORD, BYTE or Word to a fixed length String.
the string will be filled with leading zeroes to achieve the fixed length, or if too long, the lowest digits will be used.
the maximum allowed length is 20 mdigits.

for example:	dword_to_strf(123,4) = '0123' 
				dword_to_strf(123,2) = '23'
*)

(* limit N to max 20 characters *)
(* convert dword to string first and cut to length N *)
DWORD_TO_STRF := FIX(DWORD_TO_STRING(in),LIMIT(0,N,20),48,1);


(* revision history
hm	26. jan.2007	rev 1.0		
	original version

hm	29. mar. 2008	rev 1.1
	changed STRING to STRING(20)
	limit the output string to max 20 digits
*)

END_FUNCTION

// POUs/String/FIX
FUNCTION FIX : STRING(STRING_LENGTH)
VAR_INPUT
	str : STRING(STRING_LENGTH);
	L : INT;
	C : BYTE;
	M : INT;
END_VAR
VAR
	N : INT;
	SX: STRING(STRING_LENGTH);
END_VAR

(*
version 1.0	29. mar. 2008
programmer 	hugo
tested by	tobias

the function fix truncates a string at length L 
or if the string is shorter then L it will be filled with ending Spaces till its length = N.

*)

(* make sure L does not exceed the limits of a string *)
N := LIMIT(0,L,STRING_LENGTH) - LEN(str);
IF N <= 0 THEN
	(* truncate the string at length N *)
	IF M = 1 THEN
		FIX := RIGHT(str,L);
	ELSE
		FIX := LEFT(str,L);
	END_IF;
ELSIF M = 1 THEN
	(* connect fill characters at the beginning *)
	sx := FILL(C,N);
	FIX := CONCAT(sx,str);
ELSIF M = 2 THEN
	(* center str beween fill characters *)
	(* for an uneven number of fill characters, there is one more at the end *)
	sx := FILL(C,SHR(N+1,1));
	FIX := CONCAT(str,sx);
	SX := LEFT(sx,SHR(N,1));
	FIX := CONCAT(sx,FIX);
ELSE
	(* connect fill characters at the end *)
	SX := FILL(C,N);
	FIX := CONCAT(str,SX);
END_IF;


(* revision histroy
hm	29. mar. 2008	rev 1.0
	original release

*)

END_FUNCTION

// POUs/String/DWORD_TO_STRH
FUNCTION DWORD_TO_STRH : STRING(8)
VAR_INPUT
	IN : DWORD;
END_VAR
VAR
	i : INT;
	temp : BYTE;
	pt : POINTER TO BYTE;
END_VAR

(*
version 1.3	29. mar. 2008
programmer 	hugo
tested by	tobias

DWORD_TO_STRINGH converts a DWORD to a String of Hexadecimal represented by '0' .. '9' and 'A' .. 'F'.
The lowest order Character will be on the right and the high order Character on the left.

*)

(* read output adress to pointer *)
pt := ADR(DWORD_TO_STRH) + 8;
(* wirte the closing byte for the string *)
pt^:= 0;

(* write the 8 hex characters backwards *)
FOR i := 1 TO 8 DO;
	(* decrement the pointer *)
	pt := pt - 1;
	(* read the lowest order hex value *)
	temp := DWORD_TO_BYTE(in AND 16#0000000F);
	(* convert value to hex character *)
	IF temp <= 9 THEN temp := temp + 48; ELSE temp := temp + 55; END_IF;
	(* write character to output string *)
	PT^ := temp;
	(* shift in for nect hex character *)
	in := SHR(in,4);
END_FOR;


(* code beofre rev 1.2
FOR i := 1 TO 8 DO
	X := DWORD_TO_BYTE(in AND 2#1111);
	IF X <= 9 THEN X := X + 48; ELSE X := X + 55; END_IF;
	Cx := CHR(X);
	temp := CONCAT(Cx, temp);
	in := SHR(in,4);
END_FOR;
DWORD_TO_STRH := temp;
*)


(* revision history
hm	9. jun. 2007	rev 1.0		
	original version 

hm	11. sep. 2007	rev 1.1
	changed coding for compatibility with twincat, concat cannot support a function as an argument.

hm	15. dec. 2007	rev 1.2
	changed code for better performance

hm	29. mar. 2008	rev 1.3
	changed STRING to STRING(8)

*)

END_FUNCTION

// POUs/Mathematical/Geometry/ELLIPSE_A
FUNCTION ELLIPSE_A : REAL
VAR_INPUT
	R1 : REAL;
	R2 : REAL;
END_VAR


(*
version 1.1	18. oct. 2008
programmer 	hugo
tested by	oscat

ellipse_A calculates the Area of an ellipe based on the two radians R1 and R2


*)

ELLIPSE_A := math.PI * R1 * R2;

(* revision histroy
hm	16. oct 2007	rev 1.0
	original version

hm	18. oct. 2008	rev 1.1
	using math constants
*)

END_FUNCTION

// POUs/Mathematical/Geometry/ELLIPSE_C
FUNCTION ELLIPSE_C : REAL
VAR_INPUT
	R1 : REAL;
	R2 : REAL;
END_VAR


(*
version 1.2	10. mar. 2009
programmer 	hugo
tested by		oscat

ellipse_C calculates the circumference of an ellipe based on the two radians R1 and R2

*)

ELLIPSE_C := math.PI * (3.0 * (R1+R2) - SQRT((3.0 * r1 + R2) * (3.0 * r2 + r1)));

(* revision histroy
hm	16. oct 2007	rev 1.0
	original version

hm	18. oct. 2008	rev 1.1
	using math constants

hm	10. mar. 2009	rev 1.2
	changed syntax of real constants to 0.0

*)

END_FUNCTION

// POUs/Engineering/conversion/ENERGY
FUNCTION_BLOCK ENERGY
VAR_INPUT
	J : REAL;
	C : REAL;
	Wh : REAL;
END_VAR
VAR_OUTPUT
	YJ : REAL;
	YC : REAL;
	YWh : REAL;
END_VAR


(*
version 1.2	16. jan. 2010
programmer 	hugo
tested by		oscat

this function converts different energy units
any unused input can simply be left open.
different inputs connected at the same time will be added up.
*)

YJ := J + Wh * 3600.0 + C * 4.1868;
YC := YJ * 0.238845896627496;
YWh := YJ * 2.7777777778E-004;

(*
Arbeit, Energie, Joule* J 1 J = 1 N · m = 1 W · s = (1/3,6) E6 kW · h = 1 kg · m2/s2
Wärmemenge Kilowattstunde kW · h 1 kW · h = 3,6 MJ = 860 kcal
Elektronvolt eV 1 eV = 160,218 92 E21 J
Erg erg 1 erg = 1E7 J
Kalorie calorie 1 calalorie = 4,1868 J = 1,163 E3 W · h
Therm therm 1 therm = 105,50 · 106 J
*)

(* revision history

hm	27. mar. 2007	rev 1.0
	original version

hm	11. mar. 2009	rev 1.1
	improved code

hm 16. jan 2010	rev 1.2
	avoid the string cal in comments for codesys import bug


*)

END_FUNCTION_BLOCK

// POUs/Mathematical/ERF
FUNCTION ERF : REAL
VAR_INPUT
	X : REAL;
END_VAR
VAR
	x2 : REAL;
	ax2 : REAL;
END_VAR


(*
version 1.3	10. mar. 2009
programmer 	hugo
tested by		tobias

this function calculates the erf (error) function.

*)

x2 := X*X;
ax2 := 0.147 * x2 + 1.0;
ERF := SQRT(1.0 - EXP(-X2 * ((0.27323954473516 + aX2)/(ax2)))) * SGN(x);




(* revision history
hm	7. apr. 2008	rev 1.0
	original version

hm	30. jun. 2008	rev 1.1
	added type conversions to avoid warnings under codesys 3.0

hm	25. oct. 2008	rev 1.2
	new code using new algorithm

hm	10. mar. 2009	rev 1.3
	real constants updated to new systax using dot
*)

END_FUNCTION

// POUs/Mathematical/ERFC
FUNCTION ERFC : REAL
VAR_INPUT
	X : REAL;
END_VAR


(*
version 1.1	10. mar. 2009
programmer 	hugo
tested by		tobias

this function calculates the inverse erf (error) function.

*)

ERFC := 1.0 - ERF(X);

(* revision history
hm	7. apr. 2008	rev 1.0
	original version

hm	10. mar. 2009	rev 1.1
	real constants updated to new systax using dot

*)

END_FUNCTION

// POUs/Other/ESR_COLLECT
FUNCTION_BLOCK ESR_COLLECT
VAR_INPUT
	ESR_0, ESR_1, ESR_2, ESR_3, ESR_4, ESR_5, ESR_6, ESR_7 : ARRAY [0..3] OF esr_data;
	rst : BOOL;
END_VAR
VAR_IN_OUT
	pos : INT;
END_VAR
VAR_OUTPUT
	ESR_OUT : ARRAY[0..31] OF esr_data;
END_VAR
VAR CONSTANT
	max_in : INT := 3; (* max limit of input array *)
	max_out : INT := 32; (* number of elements in array *)
END_VAR
VAR
	cnt : INT := -1;
END_VAR

(*
version 1.4	1. dec. 2009
programmer 	hugo
tested by		tobias

ESR_collect collects esr data from up to 8 esr_mon modules and stroes them in an output array.
the output pos will display the position of the last element in the array. if the array is empty, pos = -1
when to buffer is read by followon modules. pos has to be reset to -1
if the array will be full, the buffer will be refilled starting at position 0.

*)

IF rst OR cnt < 0 THEN
	pos := -1;
ELSE
	FOR cnt := 0 TO max_in DO
	IF esr_0[cnt].typ > 0 THEN pos := INC1(pos, max_out); esr_out[pos] := esr_0[cnt]; END_IF;
	IF esr_1[cnt].typ > 0 THEN pos := INC1(pos, max_out); esr_out[pos] := esr_1[cnt]; END_IF;
	IF esr_2[cnt].typ > 0 THEN pos := INC1(pos, max_out); esr_out[pos] := esr_2[cnt]; END_IF;
	IF esr_3[cnt].typ > 0 THEN pos := INC1(pos, max_out); esr_out[pos] := esr_3[cnt]; END_IF;
	IF esr_4[cnt].typ > 0 THEN pos := INC1(pos, max_out); esr_out[pos] := esr_4[cnt]; END_IF;
	IF esr_5[cnt].typ > 0 THEN pos := INC1(pos, max_out); esr_out[pos] := esr_5[cnt]; END_IF;
	IF esr_6[cnt].typ > 0 THEN pos := INC1(pos, max_out); esr_out[pos] := esr_6[cnt]; END_IF;
	IF esr_7[cnt].typ > 0 THEN pos := INC1(pos, max_out); esr_out[pos] := esr_7[cnt]; END_IF;
   END_FOR;
END_IF;


(* revision history
hm	26.jan 2007	rev 1.0
	original version

hm	8. dec 2007	rev 1.1
	added reset input

ks	27. oct. 2008	rev 1.2
	optimized code for performance

ks	12. nov. 2009	rev 1.3
	output pos was not pointing to last value	

hm	1. dec. 2009	rev 1.4
	changed pos to be I/O
	reduced output array size to 32 elements
*)

END_FUNCTION_BLOCK

// POUs/Other/ESR_MON_B8
FUNCTION_BLOCK ESR_MON_B8
VAR_INPUT
	s0, s1, s2, s3, s4, s5, s6, s7 : BOOL;
	DT_in : DT;
END_VAR
VAR_INPUT CONSTANT
	a0, a1, a2, a3, a4, a5, a6, a7 : STRING(10);
END_VAR
VAR_OUTPUT
	ESR_Flag : BOOL;
END_VAR
VAR_IN_OUT
	ESR_Out: ARRAY [0..3] OF esr_data;
END_VAR
VAR
	x0, x1, x2, x3, x4, x5, x6, x7 : BOOL;
	tx: TIME;
	cnt : INT;
END_VAR

(*
version 1.3	1. dec. 2009
programmer 	hugo
tested by		tobias

ESR_mon_B8 monitores up to 8 binary inputs and reports changes with time stamd and adress label.
the module checks 8 inputs for a change and reports all changes with time and adress stamp to the output.
4 events maximum can be collected at once within the same cycle

*)

(* read system timer *)
tx := DWORD_TO_TIME(T_PLC_MS());

ESR_Flag := FALSE;
esr_out[3].typ := 0;
esr_out[2].typ := 0;
esr_out[1].typ := 0;
esr_out[0].typ := 0;
cnt := 0;


(* check if inputs have chaged and fill buffer *)
IF s0 <> X0 THEN
	esr_out[cnt].typ := 10 + BOOL_TO_BYTE(s0);
	esr_out[cnt].adress := a0;
	esr_out[cnt].DS := DT_in;
	esr_out[cnt].TS := TX;
	X0 := S0;
	cnt := cnt + 1;
	esr_flag := TRUE;
END_IF;
IF s1 <> X1 THEN
	esr_out[cnt].typ := 10 + BOOL_TO_BYTE(s1);
	esr_out[cnt].adress := a1;
	esr_out[cnt].DS := DT_in;
	esr_out[cnt].TS := TX;
	X1 := S1;
	cnt := cnt + 1;
	esr_flag := TRUE;
END_IF;
IF s2 <> X2 THEN
	esr_out[cnt].typ := 10 + BOOL_TO_BYTE(s2);
	esr_out[cnt].adress := a2;
	esr_out[cnt].DS := DT_in;
	esr_out[cnt].TS := TX;
	X2 := S2;
	cnt := cnt + 1;
	esr_flag := TRUE;
END_IF;
IF s3 <> X3 THEN
	esr_out[cnt].typ := 10 + BOOL_TO_BYTE(s3);
	esr_out[cnt].adress := a3;
	esr_out[cnt].DS := DT_in;
	esr_out[cnt].TS := TX;
	X3 := S3;
	cnt := cnt + 1;
	esr_flag := TRUE;
END_IF;
IF s4 <> X4 AND cnt < 4 THEN
	esr_out[cnt].typ := 10 + BOOL_TO_BYTE(s4);
	esr_out[cnt].adress := a4;
	esr_out[cnt].DS := DT_in;
	esr_out[cnt].TS := TX;
	X4 := S4;
	cnt := cnt + 1;
	esr_flag := TRUE;
END_IF;
IF s5 <> X5  AND cnt < 4 THEN
	esr_out[cnt].typ := 10 + BOOL_TO_BYTE(s5);
	esr_out[cnt].adress := a5;
	esr_out[cnt].DS := DT_in;
	esr_out[cnt].TS := TX;
	X5 := S5;
	cnt := cnt + 1;
	esr_flag := TRUE;
END_IF;
IF s6 <> X6  AND cnt < 4 THEN
	esr_out[cnt].typ := 10 + BOOL_TO_BYTE(s6);
	esr_out[cnt].adress := a6;
	esr_out[cnt].DS := DT_in;
	esr_out[cnt].TS := TX;
	X6 := S6;
	cnt := cnt + 1;
	esr_flag := TRUE;
END_IF;
IF s7 <> X7  AND cnt < 4 THEN
	esr_out[cnt].typ := 10 + BOOL_TO_BYTE(s7);
	esr_out[cnt].adress := a7;
	esr_out[cnt].DS := DT_in;
	esr_out[cnt].TS := TX;
	X7 := S7;
	cnt := cnt + 1;
	esr_flag := TRUE;
END_IF;

(* revision history
hm	26. jan 2007	rev 1.0
	original version

hm	17. sep 2007	rev 1.1
	replaced time() with T_PLC_MS() for compatibility reasons

hm	22. oct. 2008	rev 1.2
	optimized code

hm	1.dec. 2009	rev 1.3
	changed esr_out to be I/O

*)

END_FUNCTION_BLOCK

// POUs/Other/ESR_MON_R4
FUNCTION_BLOCK ESR_MON_R4
VAR_INPUT
	R0, R1, R2, R3 : REAL;
	DT_in : DT;
END_VAR
VAR_INPUT CONSTANT
	a0, a1, a2, a3 : STRING(10);
	s0, s1, s2, s3 : REAL;
END_VAR
VAR_OUTPUT
	ESR_Flag : BOOL;
END_VAR
VAR_IN_OUT
	ESR_Out: ARRAY [0..3] OF esr_data;
END_VAR
VAR
	p0, p1, p2, p3 : POINTER TO DWORD;
	x0, x1, x2, x3 : REAL;
	tx: TIME;
	cnt : INT;
END_VAR

(*
version 1.4	1. dec. 2009
programmer 	hugo
tested by		tobias

ESR_mon_R4 monitores up to 4 Real inputs and reports changes with time stamd and adress label.
the module checks 4 inputs for a change of more than the specified sensitivity S and reports all changes with time and adress stamp to the output.

*)

(* read system timer *)
tx := DWORD_TO_TIME(T_PLC_MS());
P0 := ADR(R0);
P1 := ADR(R1);
P2 := ADR(R2);
P3 := ADR(R3);

ESR_Flag := FALSE;
esr_out[3].typ := 0;
esr_out[2].typ := 0;
esr_out[1].typ := 0;
esr_out[0].typ := 0;
cnt := 0;

(* check if inputs have chaged and fill buffer *)
IF DIFFER(R0,  X0, S0) THEN
	esr_out[cnt].typ := 20;
	esr_out[cnt].adress := a0;
	esr_out[cnt].DS := DT_in;
	esr_out[cnt].TS := TX;
	esr_out[cnt].data[0] := Byte_of_Dword(P0^,0);
	esr_out[cnt].data[1] := Byte_of_Dword(P0^,1);
	esr_out[cnt].data[2] := Byte_of_Dword(P0^,2);
	esr_out[cnt].data[3] := Byte_of_Dword(P0^,3);
	X0 := R0;
	cnt := cnt + 1;
	esr_flag := TRUE;
END_IF;
IF differ(R1,  X1, S1) THEN
	esr_out[cnt].typ := 20;
	esr_out[cnt].adress := a1;
	esr_out[cnt].DS := DT_in;
	esr_out[cnt].TS := TX;
	esr_out[cnt].data[0] := Byte_of_Dword(P1^,0);
	esr_out[cnt].data[1] := Byte_of_Dword(P1^,1);
	esr_out[cnt].data[2] := Byte_of_Dword(P1^,2);
	esr_out[cnt].data[3] := Byte_of_Dword(P1^,3);
	X1 := R1;
	cnt := cnt + 1;
	esr_flag := TRUE;
END_IF;
IF differ(R2,  X2, S2) THEN
	esr_out[cnt].typ := 20;
	esr_out[cnt].adress := a2;
	esr_out[cnt].DS := DT_in;
	esr_out[cnt].TS := TX;
	esr_out[cnt].data[0] := Byte_of_Dword(P2^,0);
	esr_out[cnt].data[1] := Byte_of_Dword(P2^,1);
	esr_out[cnt].data[2] := Byte_of_Dword(P2^,2);
	esr_out[cnt].data[3] := Byte_of_Dword(P2^,3);
	X2 := R2;
	cnt := cnt + 1;
	esr_flag := TRUE;
END_IF;
IF DIFFER(R3,  X3, S3) THEN
	esr_out[cnt].typ := 20;
	esr_out[cnt].adress := a3;
	esr_out[cnt].DS := DT_in;
	esr_out[cnt].TS := TX;
	esr_out[cnt].data[0] := Byte_of_Dword(P3^,0);
	esr_out[cnt].data[1] := Byte_of_Dword(P3^,1);
	esr_out[cnt].data[2] := Byte_of_Dword(P3^,2);
	esr_out[cnt].data[3] := Byte_of_Dword(P3^,3);
	X3 := R3;
	cnt := cnt + 1;
	esr_flag := TRUE;
END_IF;


(* revision history
hm	26. jan 2007	rev 1.0
	original version

hm	17. sep. 2007		rev 1.1
	replaced time() with T_PLC_MS() for compatibility reasons

hm	8. dec. 2007		rev 1.2
	corrected an error while esr typ would not be set

hm	16. mar. 2008		rev 1.3
	deleted wrong conversion real_to_dword

hm	1. dec 2009		rev 1.4
	changed esr_out to be I/O

*)

END_FUNCTION_BLOCK

// POUs/Other/ESR_MON_X8
FUNCTION_BLOCK ESR_MON_X8
VAR_INPUT
	s0, s1, s2, s3, s4, s5, s6, s7 : BYTE;
	DT_in : DT;
	Mode : BYTE := 3;
END_VAR
VAR_INPUT CONSTANT
	a0, a1, a2, a3, a4, a5, a6, a7 : STRING(10);
END_VAR
VAR_OUTPUT
	ESR_Flag : BOOL;
END_VAR
VAR_IN_OUT
	ESR_Out: ARRAY [0..3] OF esr_data;
END_VAR
VAR
	x0, x1, x2, x3, x4, x5, x6, x7 : BYTE;
	tx: TIME;
	cnt : INT;
END_VAR

(*
version 1.2	1. dec. 2009
programmer 	hugo
tested by		tobias

ESR_MON_X8 is a status and error collector.
the module checks 8 status inputs for a change and reports up to 4 input changes with time and adress stamp to the output.
the mode can be 
1 for error only
2 for error and status
3 for error, status and debug
the adress label of the 8 inputs can be configured individually.
*)

(* read system timer *)
tx := DWORD_TO_TIME(T_PLC_MS());

ESR_Flag := FALSE;
esr_out[3].typ := 0;
esr_out[2].typ := 0;
esr_out[1].typ := 0;
esr_out[0].typ := 0;
cnt := 0;


(* check if inputs have chaged and fill buffer *)
IF s0 <> X0 AND ((s0 < 100) OR (S0 > 99 AND S0 < 200 AND mode >= 2) OR (S0 > 199 AND mode = 3)) THEN
	esr_out[cnt] := status_to_ESR(s0, a0, DT_in, TX);
	X0 := S0;
	cnt := cnt + 1;
	esr_flag := TRUE;
END_IF;
IF s1 <> X1 AND ((s1 < 100) OR (S1 > 99 AND S1 < 200 AND mode >= 2) OR (S1 > 199 AND mode = 3)) THEN
	esr_out[cnt] := status_to_ESR(s1, a1, DT_in, TX);
	X1 := S1;
	cnt := cnt + 1;
	esr_flag := TRUE;
END_IF;
IF s2 <> X2 AND ((s2 < 100) OR (S2 > 99 AND S2 < 200 AND mode >= 2) OR (S2 > 199 AND mode = 3)) THEN
	esr_out[cnt] := status_to_ESR(s2, a2, DT_in, TX);
	X2 := S2;
	cnt := cnt + 1;
	esr_flag := TRUE;
END_IF;
IF s3 <> X3 AND ((s3 < 100) OR (S3 > 99 AND S3 < 200 AND mode >= 2) OR (S3 > 199 AND mode = 3)) THEN
	esr_out[cnt] := status_to_ESR(s3, a3, DT_in, TX);
	X3 := S3;
	cnt := cnt + 1;
	esr_flag := TRUE;
END_IF;
IF cnt < 4 AND s4 <> X4 AND ((s4 < 100) OR (S4 > 99 AND S4 < 200 AND mode >= 2) OR (S4 > 199 AND mode = 3)) THEN
	esr_out[cnt] := status_to_ESR(s4, a4, DT_in, TX);
	X4 := S4;
	cnt := cnt + 1;
	esr_flag := TRUE;
END_IF;
IF cnt < 4 AND s5 <> X5 AND ((s5 < 100) OR (S5 > 99 AND S5 < 200 AND mode >= 2) OR (S5 > 199 AND mode = 3)) THEN
	esr_out[cnt] := status_to_ESR(s5, a5, DT_in, TX);
	X5 := S5;
	cnt := cnt + 1;
	esr_flag := TRUE;
END_IF;
IF cnt < 4 AND s6 <> X6 AND ((s6 < 100) OR (S6 > 99 AND S6 < 200 AND mode >= 2) OR (S6 > 199 AND mode = 3)) THEN
	esr_out[cnt] := status_to_ESR(s6, a6, DT_in, TX);
	X6 := S6;
	cnt := cnt + 1;
	esr_flag := TRUE;
END_IF;
IF cnt < 4 AND s7 <> X7 AND ((s7 < 100) OR (S7 > 99 AND S7 < 200 AND mode >= 2) OR (S7 > 199 AND mode = 3)) THEN
	esr_out[cnt] := status_to_ESR(s7, a7, DT_in, TX);
	X7 := S7;
	cnt := cnt + 1;
	esr_flag := TRUE;
END_IF;


(* revision history
hm	26. jan 2007		rev 1.0
	original version

hm	17. sep 2007	rev 1.1
	replaced time() with T_PLC_MS() for compatibility reasons

hm	1. dec. 2009	rev 1.2
	changed esr_out to be I/O


*)

END_FUNCTION_BLOCK

// POUs/Other/STATUS_TO_ESR
FUNCTION STATUS_TO_ESR : esr_data
VAR_INPUT
	status : BYTE;
	adress : STRING(10);
	DT_in : DT;
	TS : TIME;
END_VAR


(*
version 1.0	6 oct 2006
programmer 	hugo
tested by		tobias

status_to_esr creates esr data from a status byte.

*)

IF status < 100 THEN
	status_to_ESR.typ := 1;
ELSIF status < 200 THEN
	status_to_ESR.typ := 2;
ELSE
	status_to_ESR.typ := 3;
END_IF;
status_to_ESR.adress:= adress;
status_to_ESR.DS := DT_in;
status_to_ESR.TS := TS;
status_to_ESR.data[0] := status;

END_FUNCTION

// POUs/String/EXEC
FUNCTION EXEC : STRING(STRING_LENGTH)
VAR_INPUT
	str : STRING(STRING_LENGTH);
END_VAR
VAR
	pos: INT;
	R1: REAL;
	R2: REAL;
	operator: STRING(10);
END_VAR

(*
version 1.4	29. mar. 2008
programmer 	hugo
tested by		tobias

exec executes a mathematical term and returns the result as a string
the term can only be a simple term without brackets and only one operator
allowed operastors are: (+, -, *, /, ^, sqrt, sin, cos, tan).

*)

(* extract both numbers and operator *)
EXEC := UPPERCASE(TRIM(str));

pos := FINDB_NONUM(EXEC);
IF pos > 1 THEN R1 := STRING_TO_REAL(LEFT(EXEC,pos-1)); END_IF;
R2 := STRING_TO_REAL(RIGHT(EXEC,LEN(EXEC)-pos));
EXEC := LEFT(EXEC,pos);
pos := FINDB_NUM(EXEC);
operator := RIGHT(EXEC,LEN(EXEC) - pos);
IF operator = '' AND LEN(str) = 0 THEN
	EXEC := '';
	RETURN;
ELSIF operator = '' THEN
	EXEC := str;
	RETURN;
END_IF;
IF operator = '^' THEN
	EXEC := REAL_TO_STRING(EXPT(R1, R2));
ELSIF operator = 'SQRT' THEN
	EXEC := REAL_TO_STRING(SQRT(R2));
ELSIF operator = 'SIN' THEN
	EXEC := REAL_TO_STRING(SIN(r2));
ELSIF operator = 'COS' THEN
	EXEC := REAL_TO_STRING(COS(r2));
ELSIF operator = 'TAN' THEN
	EXEC := REAL_TO_STRING(TAN(R2));
ELSIF operator = '*' THEN
	EXEC := REAL_TO_STRING(R1 * R2);
ELSIF operator = '/' THEN
	IF R2 <> 0 THEN EXEC := REAL_TO_STRING(R1 / R2); ELSE EXEC := 'ERROR'; END_IF;
ELSIF operator = '+' THEN
	EXEC := REAL_TO_STRING(r1 + r2);
ELSIF operator = '-' THEN
	EXEC := REAL_TO_STRING(r1 - r2);
ELSE
	EXEC := 'ERROR';
END_IF;

IF EXEC = 'ERROR' THEN
	RETURN;
(* some systems deliver integer instead of real *)
ELSIF FIND(EXEC,'.') = 0 THEN
	EXEC := CONCAT(EXEC, '.0');
(* some systems deliver n. instead of n.0 ! *)
ELSIF RIGHT(EXEC,1) = '.' THEN
	EXEC := CONCAT(EXEC,'0');
END_IF;


(* revision history

hm 	6.feb 2007		rev 1.1
	cos has to be written in uppercase
	divide by 0 will return an error

hm	5. mar. 2008	rev 1.2
	add a 0 to the string if a '.' is at the end of the string

hm	20. mar. 2008	rev 1.3
	make sure the function always returns a real value in the form of x.y

hm	29. mar. 2008	rev 1.4
	changed STRING to STRING(STRING_LENGTH)
*)

END_FUNCTION

// POUs/String/TRIM
FUNCTION TRIM : STRING(STRING_LENGTH)
VAR_INPUT
	str : STRING(STRING_LENGTH);
END_VAR
VAR
	pos: INT;
END_VAR

(*
version 1.2	29. mar. 2008
programmer 	hugo
tested by	tobias

the function deletes all blanks within a string.

*)

TRIM := str;
REPEAT
	pos := FIND(trim,' ');
	IF pos > 0 THEN TRIM := REPLACE(TRIM,'',1,pos); END_IF;
UNTIL pos = 0	END_REPEAT;


(* revision histroy
hm	6.10.2006		rev 1.0
	original release

hm	20. mar. 2008	rev 1.1
	avoid to call replace with pos = 0 because some systems will produce an error

hm	29. mar. 2008	rev 1.2
	changed STRING to STRING(STRING_LENGTH)
*)

END_FUNCTION

// POUs/String/FINDB_NONUM
FUNCTION FINDB_NONUM : INT
VAR_INPUT
	str : STRING(STRING_LENGTH);
END_VAR
VAR
	pos: INT;
	pt : POINTER TO BYTE;
END_VAR

(*
version 1.3	21. oct. 2008
programmer 	hugo
tested by	oscat

findB_noNum searches str backwards and returns the last position which is not a number.
a number is characterized by a letter "0..9" or "."

*)

pt := ADR(str) + LEN(str) - 1;
FOR pos := LEN(str) TO 1 BY -1 DO;
	IF (PT^ < 48 AND PT^ <> 46) OR PT^ > 57 THEN
		FINDB_NONUM := pos;
		RETURN;
	END_IF;
	PT := PT - 1;
END_FOR;
FINDB_NONUM := 0;


(* revision history
hm	6. oct 2006		rev 1.0
	original version

hm	29. feb 2008	rev 1.1
	improved performance

hm	29. mar. 2008	rev 1.2
	changed STRING to STRING(STRING_LENGTH)

hm	21. oct. 2008	rev 1.3
	optimized code
*)

END_FUNCTION

// POUs/String/FINDB_NUM
FUNCTION FINDB_NUM : INT
VAR_INPUT
	str : STRING(STRING_LENGTH);
END_VAR
VAR
	pos: INT;
	pt : POINTER TO BYTE;
END_VAR

(*
version 1.2	29. mar. 2008
programmer 	hugo
tested by	tobias

findB_Num searches str backward and returns the last position of a number
a number is characterized by a letter "0..9" or "."

*)

pt := ADR(str) + LEN(str) - 1;
FOR pos := LEN(str) TO 1 BY -1 DO;
	IF (PT^ > 47 AND PT^ < 58) OR PT^ = 46 THEN
		FINDB_NUM := pos;
		RETURN;
	END_IF;
	PT := PT - 1;
END_FOR;
FINDB_NUM := 0;

(* revision history
hm	6. oct 2006		rev 1.0
	original version

hm	29. feb 2008	rev 1.1
	improved performance

hm	29. mar. 2008	rev 1.2
	changed STRING to STRING(STRING_LENGTH)
*)

END_FUNCTION

// POUs/Mathematical/EXPN
FUNCTION EXPN : REAL
VAR_INPUT
	X : REAL;
	N : INT;
END_VAR
VAR
	sign: BOOL;
END_VAR

(*
version 1.2	10. mar. 2009
programmer 	hugo
tested by		oscat

this function calculates X to the power of N (Y = X^N) whilke N is an integer
especially on CPU's without a floating point unit this algorythm is about 30 times faster then the IEC standard EXPT() Function

*)

sign := n.15;
N := ABS(N);
IF N.0 THEN EXPN := X; ELSE EXPN := 1.0; END_IF;
N := SHR(N,1);
WHILE N > 0 DO
   X := X * X;
   IF N.0 THEN EXPN := EXPN * X; END_IF;
   N := SHR(N,1);
END_WHILE;
IF sign THEN EXPN := 1.0 / EXPN; END_IF;



(* revision history
hm	4. dec 2007	rev 1.0
	original version

hm	22. oct. 2008	rev 1.1
	optimized code

hm	10. mar. 2009	rev 1.2
	removed nested comments
	real constants updated to new systax using dot

*)

END_FUNCTION

// POUs/Building/electrical/F_LAMP
FUNCTION_BLOCK F_LAMP
VAR_INPUT
	SWITCH : BOOL;
	DIMM : BYTE := 255;
	RST : BOOL;
END_VAR
VAR_OUTPUT
	LAMP : BYTE;
	STATUS : BYTE;
END_VAR
VAR_IN_OUT
	ONTIME : UDINT;
	CYCLES : UDINT;
END_VAR
VAR_INPUT CONSTANT
	T_NO_DIMM : UINT := 100;
	T_MAINTENANCE : UINT := 15000;
END_VAR
VAR
	runtime : ONTIME;
END_VAR

(*
version 1.2	22. oct. 2008
programmer 	hugo
tested by	oscat

F_Lamp is an interface to flourescent lamps. its main purpose is to protect flourescent lamps from dimming within the first T_NO_DIMM Time.
If Flourescent Lamps are dimmed during the first 100 hours the lifetime of the lamp is reduced dramatically.
The interface also counts ontime and cycles of the lamp for maintanance purposes.

*)

runtime(in := switch, seconds := ontime, cycles := cycles);

IF RST THEN
	ONTIME := 0;
	CYCLES := 0;
END_IF;
IF SWITCH THEN
	IF ontime < T_NO_DIMM * 3600 THEN
		LAMP := 255;
		STATUS := 111;
	ELSE
		LAMP := DIMM;
		STATUS := 112;
	END_IF;
ELSE
	LAMP := 0;
	STATUS := 110;
END_IF;


IF ontime >= T_maintenance * 3600 AND T_Maintenance > 0 THEN
	status := 120;
END_IF;



(* revision history
hm	8. feb. 2007	rev 1.1
	original version

hm	22. oct. 2008	rev 1.2
	changed use of ontime for ontime 2.0
	ontime is now in seconds not hours
*)

END_FUNCTION_BLOCK

// POUs/Mathematical/functions/F_LIN
FUNCTION F_LIN : REAL
VAR_INPUT
	X : REAL;
	A : REAL;
	B : REAL;
END_VAR


(*
version 1.0	1 sep 2006
programmer 	hugo
tested by		tobias

this function calculates the linear equation f_lin = a*x + b

*)

F_lin := A * X + B;

END_FUNCTION

// POUs/Mathematical/functions/F_LIN2
FUNCTION F_LIN2 : REAL
VAR_INPUT
	X : REAL;
	X1: REAL;
	Y1 : REAL;
	X2 : REAL;
	Y2 : REAL;
END_VAR


(*
version 1.0	1 jan 2007
programmer 	hugo
tested by		tobias

this function calculates the linear equation f_lin = a*x + b given by two points x1/y1 and x2/y2.

*)

F_LIN2 := (Y2 - Y1) / (X2 - X1) * (X - X1) + Y1;


(* revision history
hm	1. jan. 2007	rev 1.0
	original release

hm	17. dec. 2008	rev 1.1
	optimized formula

*)

END_FUNCTION

// POUs/Mathematical/functions/F_POLY
FUNCTION F_POLY : REAL
VAR_INPUT
	X : REAL;
	C : ARRAY[0..7] OF REAL;
END_VAR
VAR
	x2: REAL;
	X4 : REAL;
	X6: REAL;
END_VAR

(*
version 1.0	20. may. 2008
programmer 	hugo
tested by		tobias

this function calculates the polynom C[0] + C[1]*X^1 + C[2]*X^2 * C[3]*X^3 + C[4]*X^4 + C[5]*X^5 + C[6]*X^6 + C[7]*X^7

*)

x2 := X * X;
X4 := X2 * X2;
X6 := X4 * X2;
F_POLY := C[7] * X6 * X + C[6] * X6 + C[5] * X4 * X + C[4] * X4 + c[3] * X2*X + C[2] * X2 + C[1] * X + C[0];


(* revision history
hm		20. may. 2008		rev 1.0
	original version

*)

END_FUNCTION

// POUs/Mathematical/functions/F_POWER
FUNCTION F_POWER : REAL
VAR_INPUT
	a : REAL;
	x : REAL;
	n : REAL;
END_VAR


(*
version 1.0	1 sep 2006
programmer 	hugo
tested by		tobias

this function calculates the power equation f_power = a*x^n

*)

F_POWER := a * EXPT(X, N);

END_FUNCTION

// POUs/Mathematical/functions/F_QUAD
FUNCTION F_QUAD : REAL
VAR_INPUT
	X : REAL;
	A : REAL;
	B : REAL;
	C : REAL;
END_VAR


(*
version 1.0	1 sep 2006
programmer 	hugo
tested by		tobias

this function calculates the quadratic equation f_lin = a*x + b

*)

F_QUAD := A * X * X + B * X + C;

(* revision history

hm	1. sep. 2006
	original version

*)

END_FUNCTION

// POUs/Engineering/conversion/F_TO_C
FUNCTION F_TO_C : REAL
VAR_INPUT
	fahrenheit : REAL;
END_VAR


(*
version 1.1	11. mar. 2009
programmer 	hugo
tested BY		tobias

this FUNCTION converts fahrenheit TO celsius

*)

F_TO_C := (fahrenheit - 32.0) * 0.5555555555555;

(* revision history
hm	4. aug 2006	rev 1.0
	original version

hm	11. mar. 2009	rev 1.1
	real constants updated to new systax using dot

*)

END_FUNCTION

// POUs/Engineering/conversion/F_TO_OM
FUNCTION F_TO_OM : REAL
VAR_INPUT
	F : REAL;
END_VAR


(*
version 1.1	18. oct. 2008
programmer 	hugo
tested by	oscat

this function converts frequency to Omega F
Omega = 2*PI*F
*)

F_TO_OM := math.PI2 * F;


(* revision history
hm	22. jan. 2007	rev 1.0
	original version

hm	18. oct. 2008	rev 1.1
	unsing math constants

*)

END_FUNCTION

// POUs/Engineering/conversion/F_TO_PT
FUNCTION F_TO_PT : TIME
VAR_INPUT
	F : REAL;
END_VAR


(*
version 1.1	11. mar. 2009
programmer 	hugo
tested by		tobias

this function converts frequency to periode time  
*)

F_TO_PT := DWORD_TO_TIME(REAL_TO_DWORD(1.0 / F * 1000.0));


(* revision history

hm	4. aug. 2006	rev 1.0
	original version

hm	11. mar. 2009	rev 1.1
	real constants updated to new systax using dot

*)

END_FUNCTION

// POUs/Mathematical/FACT
FUNCTION FACT : DINT
VAR_INPUT
	X : INT;
END_VAR
VAR
	i: INT;
END_VAR

(*
version 1.4	27. 0ct. 2008
programmer 	hugo
tested by		tobias

this function calculates the factorial of x

if the input is negative or higher then 7 the output will be -1.

*)

IF X <= 5 THEN
	FACT := 1;
	FOR i := 2 TO x DO
		FACT := FACT * i;
	END_FOR;
ELSIF x <= 9 THEN
	FACT := 720;
	FOR i := 7 TO x DO
		FACT := FACT * i;
	END_FOR;
ELSIF x <= 13 THEN
	FACT := 3628800;
	FOR i := 11 TO x DO
		FACT := FACT * i;
	END_FOR;
ELSE
	FACT := -1;
END_IF;




(* revision history
hm 4.3.2007		rev 1.1
	changed a critical error where while loop was indefinite.

hm	10.12.2007	rev 1.2
	start value for i has changed to 2 for better performance

hm	10. mar 2008	rev 1.3
	changed output of fact to dint to allow bigger values

hm	27. oct. 2008	rev 1.4
	optimized code
*)

END_FUNCTION

// POUs/Engineering/signal processing/FADE
FUNCTION_BLOCK FADE
VAR_INPUT
	IN1 : REAL;
	IN2 : REAL;
	F : BOOL;
	TF : TIME;
	rst : BOOL;
END_VAR
VAR_OUTPUT
	Y : REAL;
END_VAR
VAR
	rmx : RMP_W;
END_VAR

(*
version 1.3	24. jan. 2009
programmer 	oscat
tested BY		oscat

FADE is used to crossfade between the inputs IN1 and IN2. The fade_over time is specified with TF.
When F = TRUE then Y = IN2 after the time TF, and when F = FALSE then Y = IN1.

*)

rmx(rst := rst AND NOT F, set := rst AND F, pt := TF, up := F);
Y := (in2 - In1) / 65535.0 * WORD_TO_REAL(rmx.out) + in1;


(* code for rev 1.1
IF rst THEN
	rmx(set := F, rst := NOT F);
ELSIF F AND (NOT rmx.high) THEN
	rmx(PT := TF, UP := TRUE, e := TRUE, rst := FALSE, set := FALSE);
ELSIF (NOT F) AND (NOT rmx.low) THEN
	rmx(PT := TF, UP := FALSE, e := TRUE, rst := FALSE, set := FALSE);
ELSE
	rmx(e := FALSE, rst := FALSE, set := FALSE);
END_IF;
Y := (WORD_TO_REAL(rmx.out) * in1 + WORD_TO_REAL(FF - rmx.out) * IN2) / FF;
*)


(* revision history
hm	26. dec 2007	rev 1.0
	original version

hm	18. oct. 2008	rev 1.1
	improved performance
	changed calls for rmp_w because rmp_w has chaged

hm	17. dec. 2008	rev 1.2
	function of input f was inverted

hm	24. jan. 2009	rev 1.3
	delted unused var FF
*)

END_FUNCTION_BLOCK

// POUs/Engineering/signal generators/RMP_W
FUNCTION_BLOCK RMP_W
VAR_INPUT
	SET : BOOL;
	PT : TIME;
	E : BOOL := TRUE;
	UP : BOOL := TRUE;
	RST : BOOL;
END_VAR
VAR_OUTPUT
	out : WORD;
	busy : BOOL;
	high : BOOL;
	low : BOOL;
END_VAR
VAR
	rmp : _RMP_W;
END_VAR

(*
version 2.0	23. oct. 2008
programmer 	oscat
tested BY	oscat

this ramp generator generates a Word wide ramp with 65535 steps
the generator has an asynchronous set and reset
the ramp is controlled by PT which is the total ramp time for a full sweep from 0..65535
an UD input controlls the direction Up or Down and the E input enables the ramp generation
a busy output indicates that the ramp is running, busy false means output is stable.
the outputs low and high will be true when the output has reached its max or min value.
*)

(* generate ramp *)
rmp(dir := UP, E := E, TR := PT, rmp := out);

(* set or reset operation *)
IF RST THEN
	out := 0;
ELSIF SET THEN
	out := 65535;
END_IF;

(* checks for outputs stable and reset or set busy flag *)
low := out = 0;
high := out = 65535;
busy := NOT (low OR high) AND E;


(* revision history:

hm 4.10.2006		rev 1.1
	added the busy output which signals that the ramp is running.

hm 22.1.2007		rev 1.2
	deleted unused variable step

hm	17.9.2007		rev 1.3
	replaced time() with t_plc_ms() for compatibility reasons

hm	28. sep 2007	rev 1.4
	added outputs on and off
	busy is now disabled while en is false
	new coding for higher accuracy and performance

hm	5. oct 2007	rev 1.5
	added statements to allow for PT to be t#0s output jumps to max or min immediately

hm	2. dec 2007	rev 1.6
	corrected an error in calculation of step response

hm	25. dec 2007	rev 1.7
	corrected an error while step response was too slow for fast rise times

hm	16. oct. 2008	rev 1.8
	improved performance

hm	18. oct. 2008	rev 1.9
	renamed inout EN to E for compatibility reasons

hm	23. oct. 2008	rev 2.0
	new code using _RMP_W
*)

END_FUNCTION_BLOCK

// POUs/Logic/FF edge triggered/FF_D2E
FUNCTION_BLOCK FF_D2E
VAR_INPUT
	D0 : BOOL;
	D1 : BOOL;
	CLK : BOOL;
	RST : BOOL;
END_VAR
VAR_OUTPUT
	Q0 : BOOL;
	Q1 : BOOL;
END_VAR
VAR
	edge : BOOL;
END_VAR

(*
version 1.3	14. mar. 2009
programmer 	hugo
tested by		oscat

dual D-type flip flop with reset and rising clock trigger

*)

IF rst THEN
	Q0 := FALSE;
	Q1 := FALSE;
ELSIF clk AND NOT edge THEN
	Q0 := D0;
	Q1 := D1;
END_IF;
edge := CLK;

(* revision history
hm	25. dec 2007	rev 1.0
	original version

hm	27. dec 2007	rev 1.1
	changed code for better performance

hm	30. oct. 200	rev 1.2
	deleted unnecessary init with 0

hm	14. mar. 2009	rev 1.3
	removed double assignments

*)

END_FUNCTION_BLOCK

// POUs/Logic/FF edge triggered/FF_D4E
FUNCTION_BLOCK FF_D4E
VAR_INPUT
	D0 : BOOL;
	D1 : BOOL;
	D2 : BOOL;
	D3 : BOOL;
	CLK : BOOL;
	RST : BOOL;
END_VAR
VAR_OUTPUT
	Q0 : BOOL;
	Q1 : BOOL;
	Q2 : BOOL;
	Q3 : BOOL;
END_VAR
VAR
	edge : BOOL;
END_VAR


(*
version 1.3	14. mar. 2009
programmer 	hugo
tested by		oscat

quad D-type flip flop with reset and rising clock trigger

*)

IF rst THEN
	Q0 := FALSE;
	Q1 := FALSE;
	Q2 := FALSE;
	Q3 := FALSE;
ELSIF clk AND NOT edge THEN
	Q0 := D0;
	Q1 := D1;
	Q2 := D2;
	Q3 := D3;
END_IF;
edge := CLK;

(* revision history
hm	4. aug 2006	rev 1.0
	original version

hm	27. dec 2007	rev 1.1
	changed code for better performance

hm	30. oct. 200	rev 1.2
	deleted unnecessary init with 0

hm	14. mar. 2009	rev 1.3
	removed double assignments

*)

END_FUNCTION_BLOCK

// POUs/Logic/FF edge triggered/FF_DRE
FUNCTION_BLOCK FF_DRE
VAR_INPUT
	SET : BOOL;
	D : BOOL;
	CLK : BOOL;
	RST : BOOL;
END_VAR
VAR_OUTPUT
	Q : BOOL;
END_VAR
VAR
	edge : BOOL;
END_VAR


(*
version 1.2	30. oct. 2008
programmer 	hugo
tested by	oscat

D-type flip flop with set, reset and rising clock trigger

*)

IF rst OR set THEN
	Q := NOT rst;
ELSIF clk AND NOT edge THEN
	Q := D;
END_IF;
edge := CLK;

(* revision history
hm	4. aug 2006		rev 1.0
	original version

hm	27. dec 2007	rev 1.1
	changed code for better performance

hm	30. oct. 2008	rev 1.2
	optimized performance
*)

END_FUNCTION_BLOCK

// POUs/Logic/FF edge triggered/FF_JKE
FUNCTION_BLOCK FF_JKE
VAR_INPUT
	SET : BOOL;
	J : BOOL;
	CLK : BOOL;
	K : BOOL;
	RST : BOOL;
END_VAR
VAR_OUTPUT
	Q : BOOL;
END_VAR
VAR
	edge : BOOL;
END_VAR


(*
version 1.2	30. oct. 2008
programmer 	hugo
tested by	oscat

JK-type flip flop with set, reset and rising clock trigger
set and reset are asynchron while the FF is rising edge triggered
J=0 and K=0 and CLK >>> no action
J=1 and K=0 and CLK >>> output = 1
J=0 and K=1 and CLK >>> output = 0
J=1 and K=1 and CLK >>> toggle output


*)

IF rst OR set THEN
	Q := NOT rst;
ELSIF clk AND NOT edge THEN
	IF J XOR K THEN Q := J;
	ELSE Q := K XOR Q;
	END_IF;
END_IF;
edge := CLK;

(* revision history
hm	4. aug 2006		rev 1.0
	original version

hm	27. dec 2007	rev 1.1
	changed code for better performance

hm	30. oct. 2008	rev 1.2
	optimized performance
*)

END_FUNCTION_BLOCK

// POUs/Logic/FF edge triggered/FF_RSE
FUNCTION_BLOCK FF_RSE
VAR_INPUT
	CS : BOOL;
	CR : BOOL;
	RST : BOOL;
END_VAR
VAR_OUTPUT
	Q : BOOL;
END_VAR
VAR
	es, er : BOOL;
END_VAR

(*
version 1.0	16. jul. 2008
programmer 	hugo
tested by	oscat

this is a rising edge triggered rs flip flop
a rising edge on CS sets Q = TRUE and a rising edge on CR sets Q = FALSE.
CR has priority over CS.

*)

IF rst THEN
	(* asynchronous reset *)
	Q := FALSE;
ELSIF CR AND NOT er THEN
	(* rising edge on CR *)
	Q := FALSE;
ELSIF CS AND NOT es THEN
	(* rising edge on CS *)
	Q := TRUE;
END_IF;

es := CS;
er := CR;

(* revision history

hm	16. jul. 2008	rev 1.0
	original version

*)

END_FUNCTION_BLOCK

// POUs/Mathematical/FIB
FUNCTION FIB : DINT
VAR_INPUT
	X : INT;
END_VAR
VAR
	t1, t2: DINT;
END_VAR

(*
version 1.3	26. mar. 2008
programmer 	hugo
tested by		tobias

this function calculates the fibonacci sequence

*)

IF X < 0 OR X > 46 THEN
	FIB := -1;
ELSIF x < 2 THEN
	FIB := X;
	RETURN;
ELSE
	(* the fibonacci number is the sum of the two suceeding fibonaci numbers *)
	(* we store the numbers alternatively in t1 and t2 depending on pt *)
	t2 := 1;
	WHILE X > 3 DO
		X := X-2;
		t1 := t1 + t2;
		t2 := t1 + t2;
	END_WHILE;
	IF X > 2 THEN t1 := t1 + t2; END_IF;
	fib := t1 + t2;
END_IF;

(* alternative code for very big numbers

IF X < 31 THEN
	fib := 0.4472136 * (expn(1.618034,X) - expn(-0.618034,X));
ELSE
	fib := 0.4472133 * expn(1.618034,X);
END_IF;

*)

(* revision history
hm		27. dec 2007	rev 1.0
	original version

hm		2. jan 2008	rev 1.1
	deleted unused variable pt

hm		10. mar 2008	rev 1.2
	changed output to dint instead of real

hm		26. mar. 2008	rev 1.3
	function now returns -1 for input < 0 or > 46

*)

END_FUNCTION

// POUs/Logic/memory/FIFO_16
FUNCTION_BLOCK FIFO_16
VAR_INPUT
	Din : DWORD;
	E : BOOL := TRUE;
	RD : BOOL;
	WD : BOOL;
	RST : BOOL;
END_VAR
VAR_OUTPUT
	Dout : DWORD;
	EMPTY : BOOL := TRUE;
	FULL : BOOL;
END_VAR
VAR
	fifo : ARRAY[0..n] OF DWORD;
	pr : INT;
	pw : INT;
END_VAR
VAR CONSTANT
	n : INT := 16;	(* changing this value will chage the number of stored elements in the fifo *)
END_VAR


(*
version 2.0	24. jul. 2009
programmer 	hugo
tested by		oscat

16 Dword FIFO memory
*)

IF RST THEN
	pw := pr;
	FULL := FALSE;
	EMPTY := TRUE;
	Dout := 0;
ELSIF E THEN
	IF NOT EMPTY AND RD THEN
		Dout := fifo[pr];
		pr := INC1(pr,n);
		EMPTY := pr = pw;
		FULL := FALSE;
	END_IF;
	IF NOT FULL AND WD THEN
		fifo[pw] := Din;
		pw := INC1(pw,n);
		FULL := pw = pr;
		EMPTY := FALSE;
	END_IF;
END_IF;


(* revision history

hm	4. aug. 2006	rev 1.0
	original version

hm	19. feb 2008	rev 1.1
	performance improvements

hm	17. oct. 2008	rev 1.2
	improved performance

ks	27. oct. 2008	rev 1.3
	optimized coding

hm	14. mar. 2009	rev 1.4
	removed double assignments

hm 24. jul. 2009	rev 2.0
	chaged inputs E and WR to E, WD and WR
	allow read and write in one cycle

*)

END_FUNCTION_BLOCK

// POUs/Logic/memory/FIFO_32
FUNCTION_BLOCK FIFO_32
VAR_INPUT
	Din : DWORD;
	E : BOOL := TRUE;
	RD : BOOL;
	WD : BOOL;
	RST : BOOL;
END_VAR
VAR_OUTPUT
	Dout : DWORD;
	EMPTY : BOOL := TRUE;
	FULL : BOOL;
END_VAR
VAR
	fifo : ARRAY[0..n] OF DWORD;
	pr : INT;
	pw : INT;
END_VAR
VAR CONSTANT
	n : INT := 32;	(* changing this value will chage the number of stored elements in the fifo *)
END_VAR

(*
version 2.0	24. jul. 2009
programmer 	hugo
tested by		oscat

32 Dword FIFO memory
*)

IF RST THEN
	pw := pr;
	FULL := FALSE;
	EMPTY := TRUE;
	Dout := 0;
ELSIF E THEN
	IF NOT EMPTY AND RD THEN
		Dout := fifo[pr];
		pr := INC1(pr,n);
		EMPTY := pr = pw;
		FULL := FALSE;
	END_IF;
	IF NOT FULL AND WD THEN
		fifo[pw] := Din;
		pw := INC1(pw,n);
		FULL := pw = pr;
		EMPTY := FALSE;
	END_IF;
END_IF;

(* revision history
hm	4. aug. 2006	rev 1.0
	original version

hm	19. feb 2008	rev 1.1
	performance improvements

hm	17. oct. 2008	rev 1.2
	improved performance

ks	27. oct. 2008 rev 1.3
	improved code

hm	14. mar. 2009	rev 1.4
	removed double assignments

hm 24. jul. 2009	rev 2.0
	chaged inputs E and WR to E, WD and WR
	allow read and write in one cycle

*)

END_FUNCTION_BLOCK

// POUs/Engineering/signal processing/FILTER_DW
FUNCTION_BLOCK FILTER_DW
VAR_INPUT
	X : DWORD;
	T : TIME;
END_VAR
VAR_OUTPUT
	Y : DWORD;
END_VAR
VAR
	last : DWORD;
	tx: DWORD;
	init: BOOL;
	Yi : REAL;
END_VAR

(*
version 1.1	3. nov. 2008
programmer 	hugo
tested by		oscat

FILTER_DW is an low pass filter with a programmable time T used for DWORD format.
 
*)

(* read system time *)
tx := T_PLC_MS();

(* startup initialisation *)
IF NOT init OR T = t#0s THEN
	init := TRUE;
	Yi := DWORD_TO_REAL(X);
ELSE
	Yi := Yi + (DWORD_TO_REAL(X) - DWORD_TO_REAL(Y)) * DWORD_TO_REAL(tx - last) / TIME_TO_REAL(T);
END_IF;
last := tx;

Y := REAL_TO_DWORD(Yi);



(*
hm 10. oct. 2008	rev 1.0
	original version

hm	3. nov. 2008	REV 1.1
	corrected an overflow problem
*)

END_FUNCTION_BLOCK

// POUs/Engineering/signal processing/FILTER_I
FUNCTION_BLOCK FILTER_I
VAR_INPUT
	X : INT;
	T : TIME;
END_VAR
VAR_OUTPUT
	Y : INT;
END_VAR
VAR
	Yi : DINT;
	last : DWORD;
	tx: DWORD;
	init: BOOL;
END_VAR

(*
version 1.0	8. nov. 2008
programmer 	hugo
tested by	oscat

FILTER_I is a low pass filter with a programmable time T used for INT format.
 
*)

(* read system time *)
tx := T_PLC_MS();

(* startup initialisation *)
IF NOT init OR T = t#0s THEN
	init := TRUE;
	Yi := INT_TO_DINT(X) * 1000;
ELSE
	(* to increase accuracy of the filter we calculate internal Yi wich is Y * 1000 *)
	Yi := Yi + INT_TO_DINT(X - Y) * DWORD_TO_DINT(tx - last) * 1000 / TIME_TO_DINT(T);
END_IF;
last := tx;
Y := DINT_TO_INT(yi / 1000);



(*
hm 8. nov. 2008	rev 1.0
	original version

*)

END_FUNCTION_BLOCK

// POUs/Engineering/signal processing/FILTER_MAV_DW
FUNCTION_BLOCK FILTER_MAV_DW
VAR_INPUT
	X : DWORD;
	N : UINT;
	RST : BOOL;
END_VAR
VAR_OUTPUT
	Y : DWORD;
END_VAR
VAR
	init: BOOL;
	buffer : ARRAY[0..31] OF DWORD;
	i: INT;
END_VAR
VAR
	tmp: INT;
END_VAR

(*
version 1.3	23. feb. 2009
programmer 	hugo
tested by		oscat

FILTER_MAV_DW is a moving average filter with programmable length N for DWORD Data.
 
*)

(* limit N to size of buffer *)
N := MIN(N, 32);

(* startup initialisation *)
IF NOT init OR rst OR N = 0 THEN
	init := TRUE;
	tmp := UINT_TO_INT(N)-1;
	FOR i := 0 TO tmp DO
		buffer[i] := X;
	END_FOR;
	Y := X;
ELSE
	tmp := UINT_TO_INT(N);
	i := INC1(i, tmp);
	Y := Y + (X - buffer[i]) / N;
	buffer[i] := X;
END_IF;




(*
hm 13. oct. 2008	rev 1.0
	original version

hm	27. oct. 2008	rev 1.1
	added typecast to avoid warnings

hm	24. nov. 2008	rev 1.2
	added typecasts to avoid warnings
	avoid divide by 0 if N = 0

hm	23. feb. 2009	rev 1.3
	limit N to max array size

*)

END_FUNCTION_BLOCK

// POUs/Engineering/signal processing/FILTER_MAV_W
FUNCTION_BLOCK FILTER_MAV_W
VAR_INPUT
	X : WORD;
	N : UINT;
	RST : BOOL;
END_VAR
VAR_OUTPUT
	Y : WORD;
END_VAR
VAR
	init: BOOL;
	buffer : ARRAY[0..31] OF WORD;
	i: INT;
END_VAR
VAR
	tmp : INT;
END_VAR

(*
version 1.3	23. feb. 2009
programmer 	hugo
tested by		oscat

FILTER_MAV_W is a moving average filter with programmable length N for WORD Data.
 
*)

(* limit N to size of buffer *)
N := MIN(N, 32);

(* startup initialisation *)
IF NOT init OR rst OR N = 0 THEN
	init := TRUE;
	tmp := UINT_TO_INT(N) - 1;
	FOR i := 0 TO tmp DO
		buffer[i] := X;
	END_FOR;
	Y := X;
ELSE
	tmp := UINT_TO_INT(N);
	i := INC1(i, tmp);
	Y := Y + (X - buffer[i]) / N;
	buffer[i] := X;
END_IF;



(*
hm 13. oct. 2008	rev 1.0
	original version

hm	18. oct. 2008	rev 1.1
	added typecast to avoid warnings

hm	24. nov. 2008	rev 1.2
	added typecasts to avoid warnings
	avoid devide by 0 if N = 0

hm	23. feb. 2009	rev 1.3
	limit N to max array size

*)

END_FUNCTION_BLOCK

// POUs/Engineering/signal processing/FILTER_W
FUNCTION_BLOCK FILTER_W
VAR_INPUT
	X : WORD;
	T : TIME;
END_VAR
VAR_OUTPUT
	Y : WORD;
END_VAR
VAR
	last : DWORD;
	tx: DWORD;
	init: BOOL;
	tmp: DWORD;
END_VAR

(*
version 1.2	25. jan. 2011
programmer 	hugo
tested by	oscat

FILTER_W is an low pass filter with a programmable time T used for WORD format.
 
*)

(* read system time *)
tx := T_PLC_MS();

(* startup initialisation *)
IF NOT init OR T = T#0s THEN
	init := TRUE;
	last := tx;
	Y := X;
ELSIF Y = X THEN
	last := tx;
ELSE
	tmp :=  WORD_TO_DWORD(X - Y) * (tx - last) / TIME_TO_DWORD(T);
	IF tmp <> 0 THEN
		Y := DINT_TO_WORD(WORD_TO_DINT(Y) + DWORD_TO_DINT(tmp));
		last := tx;
	END_IF;
END_IF;

(*
hm 10. oct. 2008	rev 1.0
	original version

hm	3. nov. 2008	rev 1.1
	fixed overflow problem in formula

hm	25. jan. 2011	rev 1.2
	fixed error in formula
*)

END_FUNCTION_BLOCK

// POUs/Engineering/signal processing/FILTER_WAV
FUNCTION_BLOCK FILTER_WAV
VAR_INPUT
	X : REAL;
	W : ARRAY[0..15] OF REAL;
	RST : BOOL;
END_VAR
VAR_OUTPUT
	Y : REAL;
END_VAR
VAR
	init: BOOL;
	buffer : ARRAY[0..15] OF REAL;
	i: INT;
	n: INT;
END_VAR

(*
version 1.2	10. mar. 2009
programmer 	hugo
tested by		oscat

FILTER_WAV is a moving average filter with programmable length N for DWORD Data.

*)

(* startup initialisation *)
IF NOT init OR rst THEN
	init := TRUE;
	FOR i := 0 TO 15 DO
		buffer[i] := X;
	END_FOR;
	i := 15;
	Y := X;
ELSE
	i := INC1(i, 16);
	buffer[i] := X;
END_IF;

(* calculate the weighted average *)
Y := 0.0;
FOR n := 0 TO 15 DO
	Y := buffer[i] * W[n] + Y;
	i := DEC1(i, 16);
END_FOR;


(*
hm 	14. oct. 2008	rev 1.0
	original version

hm	27. oct. 2008	rev 1.1
	changed _DEC and _INC to DEC1 and INC1

hm	10. mar. 2009	rev 1.2
	real constants updated to new systax using dot

*)

END_FUNCTION_BLOCK

// POUs/String/FIND_CHAR
FUNCTION FIND_CHAR : INT
VAR_INPUT
	str : STRING(STRING_LENGTH);
	pos : INT;
END_VAR
VAR
	i: INT;
	pt : POINTER TO ARRAY[1..255] OF BYTE;
	stop: INT;
	X: BYTE;
END_VAR

(*
version 1.3	21. oct. 2008
programmer 	hugo
tested by	tobias

find_char searches str and returns the starting position of the first character that is not a control character.
control characters are the ascii character 00 .. 31 and 127

*)

pt := ADR(str);
stop := LEN(str);
FOR i := MAX(pos,1) TO stop DO;
	X := pt^[i];
	IF X > 31 AND ((setup.EXTENDED_ASCII AND X <> 127) OR (NOT setup.EXTENDED_ASCII AND X < 127)) THEN
		FIND_CHAR := i;
		RETURN;
	END_IF;
END_FOR;
FIND_CHAR := 0;


(* revision history
hm	29. feb 2008	rev 1.0
	original version

hm	26. mar. 2008	rev 1.1
	char will now accept extended ascii

hm	29. mar. 2008	rev 1.2
	changed STRING to STRING(STRING_LENGTH)

hm	21. oct. 2008	rev 1.3
	changes setup constants
	optimized code
*)

END_FUNCTION

// POUs/String/FIND_CTRL
FUNCTION FIND_CTRL : INT
VAR_INPUT
	str : STRING(STRING_LENGTH);
	pos : INT;
END_VAR
VAR
	i: INT;
	pt : POINTER TO ARRAY[1..255] OF BYTE;
	stop: INT;
	x: BYTE;
END_VAR

(*
version 1.2	29. mar. 2008
programmer 	hugo
tested by		tobias

find_ctrl searches str and returns the starting position of a control character
control characters are the ascii character 00 .. 31 and 127.

*)

pt := ADR(str);
stop := LEN(str);
FOR i := MAX(pos,1) TO stop DO;
	x := PT^[I];
	IF x < 32 OR X = 127 THEN
		FIND_CTRL := i;
		RETURN;
	END_IF;
END_FOR;
FIND_CTRL := 0;


(* revision history
hm	29. feb 2008	rev 1.0
	original version

hm	26. mar. 2008	rev 1.1
	character 127 is now recognized as control

hm	29. mar. 2008	rev 1.2
	changed STRING to STRING(STRING_LENGTH)
*)

END_FUNCTION

// POUs/String/FIND_NONUM
FUNCTION FIND_NONUM : INT
VAR_INPUT
	str : STRING(STRING_LENGTH);
	pos : INT;
END_VAR
VAR
	i: INT;
	pt : POINTER TO ARRAY[1..255] OF BYTE;
	end: INT;
	X: BYTE;
END_VAR

(*
version 1.3	21. oct. 2008
programmer 	hugo
tested by	tobias

find_noNum searches str and returns the first position which is not a number.
a number is characterized by a letter "0..9" or "."

*)

pt := ADR(str);
end := LEN(str);
FOR i := MAX(pos,1) TO end DO;
	X := pt^[i];
	IF (X < 48 AND X <> 46) OR X > 57 THEN
		FIND_NONUM := i;
		RETURN;
	END_IF;
END_FOR;
FIND_NONUM := 0;


(* revision history
hm	6. oct. 2006	rev 1.0
	original version

hm	29. feb 2008	rev 1.1
	added input pos to start search at position

hm	29. mar. 2008	rev 1.2
	changed STRING to STRING(STRING_LENGTH)

hm	21. oct. 2008	rev 1.3
	optimized code

*)

END_FUNCTION

// POUs/String/FIND_NUM
FUNCTION FIND_NUM : INT
VAR_INPUT
	str : STRING(STRING_LENGTH);
	pos : INT;
END_VAR
VAR
	i : INT;
	pt : POINTER TO ARRAY[1..255] OF BYTE;
	stop : INT;
	X: BYTE;
END_VAR

(*
version 1.2	29. mar. 2008
programmer 	hugo
tested by		tobias

find_Num searches str and returns the starting position of a number
a number is characterized by a letter "0..9" or "."

*)

pt := ADR(str);
stop := LEN(str);
FOR i := MAX(pos,1) TO stop DO;
	X := pt^[i];
	IF (X > 47 AND X < 58) OR X = 46 THEN
		FIND_NUM := i;
		RETURN;
	END_IF;
END_FOR;
FIND_NUM := 0;


(* revision history
hm	6. oct. 2006	rev 1.0
	original version

hm	29. feb 2008	rev 1.1
	added input pos to start search at position

hm	29. mar. 2008	rev 1.2
	changed STRING to STRING(STRING_LENGTH)

*)

END_FUNCTION

// POUs/String/FINDB
FUNCTION FINDB : INT
VAR_INPUT
	str1 : STRING(STRING_LENGTH);
	str2 : STRING(STRING_LENGTH);
END_VAR
VAR
	pos: INT;
	length: INT;
END_VAR

(*
version 1.3	29. mar. 2008
programmer 	hugo
tested by		tobias

the function find searches an str1 for the presence of str2 and returns the first position of str1 of the last presence in instring.
the function is similar to find except it searches from the right to left.
 a 0 is returned if the string is not found.

*)

length := LEN(str2);
FOR pos := LEN(str1) - length + 1 TO 1 BY -1 DO
	IF MID(str1,length,pos) = str2 THEN
		FindB := pos;
		RETURN;
	END_IF;
END_FOR;
FindB := 0;

(* revision history
hm	6. oct 2006		rev 1.0
	original version

hm	15 dec 2007		rev 1.1
	changed code for better performance

hm	29. feb 2008	rev 1.2
	added findb := 0 for compatibility reasons

hm	29. mar. 2008	rev 1.3
	changed STRING to STRING(STRING_LENGTH)
*)

END_FUNCTION

// POUs/String/FINDP
FUNCTION FINDP : INT
VAR_INPUT
	str : STRING(STRING_LENGTH);
	src : STRING(STRING_LENGTH);
	pos: INT;
END_VAR
VAR
	i: INT;
	ls: INT;
	lx: INT;
	stp: INT;
END_VAR

(*
version 1.2	29. mar. 2008
programmer 	hugo
tested by	tobias

the function findP searches a string str for the occurence of src beginning at the position pos.

*)

ls := LEN(str);
lx := LEN(src);
IF ls < lx OR lx = 0 THEN RETURN; END_IF;
stp := ls - lx + 1;
FOR i := MAX(pos,1) TO stp DO
	IF MID(str,lx,i) = src THEN
		FINDP := i;
		RETURN;
	END_IF;
END_FOR;
FINDP := 0;

(* revision histroy
hm	4. feb. 2008	rev 1.0
	original release

hm	29. feb 2008	rev 1.1
	ADDED MAX(pos,1) in loop initialization

hm	29. mar. 2008	rev 1.2
	changed STRING to STRING(STRING_LENGTH)
*)

END_FUNCTION

// POUs/String/FLOAT_TO_REAL
FUNCTION FLOAT_TO_REAL : REAL
VAR_INPUT
	FLT : STRING(20);
END_VAR
VAR
	pt : POINTER TO ARRAY[1..20] OF BYTE;
	i: INT;
	X: BYTE;
	sign: INT := 1;
	stop: INT;
	tmp: DINT;
	d : INT;
END_VAR

(*
version 1.3	23. oct. 2008
programmer 	hugo
tested by	oscat

FLOAT_TO_REAL converts a string to a REAL.
the function ignores all wrong characters.
the comma can be , or .
the exponent has to start with capital E or lowercase e .


*)

pt := ADR(FLT);
stop := LEN(FLT);

(* we first check for sign and exit if first number or dot is reached *)
FOR i := 1 TO stop DO
	X := pt^[i];
	IF X > 47 AND X < 58 OR X = 46 THEN
		EXIT;
	ELSIF X = 45 THEN
		(* code 45 is sign *)
		sign := -1;
	END_IF;
END_FOR;

(* now we scan numbers till end or dot or E is reached *)
FOR i := i TO stop DO
	X := pt^[i];
	IF X = 44 OR X = 46 OR X = 69 OR X = 101 THEN
		EXIT;
	(* calculate the value of the digit *)
	ELSIF X > 47 AND x < 58 THEN
		tmp := tmp * 10 + X - 48;
	END_IF;
END_FOR;

(* process the portion after the comma if comma or dot is reached exit if exponent starts *)
IF x = 44 OR X = 46 THEN
	FOR i := i + 1 TO stop DO
		X := pt^[i];
		IF X = 69 OR X = 101 THEN
			EXIT;
		ELSIF x > 47 AND x < 58 THEN
			tmp := tmp * 10 + X - 48;
			d := d - 1;
		END_IF;
	END_FOR;
END_IF;

(* process exponent if present *)
IF X = 69 OR X = 101 THEN
	d := d + DEC_TO_INT(RIGHT(FLT, stop - i));
END_IF;

FLOAT_TO_REAL :=  EXPN(10, d) * DINT_TO_REAL(TMP * SIGN);




(* revision histroy
hm	22. jun. 2008	rev 1.0
	original release

hm	2. oct. 2008	rev 1.1
	fixed an error, characters 8 and 9 would not be converted

hm	22. oct. 2008	rev 1.2
	last fix was not done correctly

hm	23. oct. 2008	rev 1.3
	optimzed code
*)

END_FUNCTION

// POUs/Engineering/automation/FLOW_CONTROL
 FUNCTION_BLOCK FLOW_CONTROL
VAR_INPUT
	IN : BOOL;
	REQ : BOOL;
	ENQ : BOOL;
	RST : BOOL;
END_VAR
VAR_INPUT CONSTANT
	T_AUTO : TIME := T#1h;
	T_DELAY : TIME := T#23h;
END_VAR
VAR_OUTPUT
	Q : BOOL;
	STATUS : BYTE;
END_VAR
VAR
	timer : TP_1D;
END_VAR


(*
version 1.0	28. jun. 2008
programmer 	hugo
tested by	oscat

FLOW_CONTROL switches a valves depending on the input in.
flow control also limits the maximum ontime of the valve and controls pressure on the output side.

*)

STATUS := 100;
IF RST THEN
	Q := FALSE;
	timer(rst := TRUE);
	timer.RST := FALSE;
	STATUS := 103;
ELSIF ENQ THEN
	IF IN THEN
		status := 101;
	END_IF;
	IF REQ THEN
		(* timer will generate a timed pulse after TP goes high *)
		timer.PT1 := T_AUTO;
		timer.PTD := T_DELAY;
		timer.IN := TRUE;
		STATUS := 102;
	END_IF;
END_IF;


(* set output and run timer *)
timer();
timer.IN := FALSE;
Q := (IN AND ENQ) OR timer.Q;



(* revision history
hm 	28. jun. 2008 	rev 1.0
	original version

*)

END_FUNCTION_BLOCK

// POUs/Logic/generators/TP_1D
FUNCTION_BLOCK TP_1D
VAR_INPUT
	IN : BOOL;
	PT1 : TIME;
	PTD : TIME;
	RST : BOOL;
END_VAR
VAR_OUTPUT
	Q : BOOL;
	W : BOOL;
END_VAR
VAR
	tx : TIME;
	start: TIME;
	ix: BOOL;
END_VAR


(*
version 1.0	28. jun. 2008
programmer 	hugo
tested by	oscat

TP_1D generates a pulse every time it is calles with in := TRUE.
the module will reset IN by itself so no clearing of in is necessary.
in addition the timer can be cleared asynchronously with rst.
also the rst input is cleared by the module itself.
the timer can be retriggered as often as necessary. it will count PT from the last trigger.
after the time PT1 is elapsed, the timer blocks itself for PT2 and only allow new sequences after PT2 has elapsed.


*)

(* read system timer *)
tx := DWORD_TO_TIME(T_PLC_MS());

IF RST THEN
	Q := FALSE;
	rst := FALSE;
	W := FALSE;
ELSIF W THEN
	IF tx - start >= PTD THEN
		W := FALSE;
	END_IF;
ELSIF IN AND NOT ix THEN
	Q := TRUE;
	start := tx;
	in := FALSE;
ELSIF tx - start >= PT1 THEN
	Q := FALSE;
	W := TRUE;
	start := tx;
END_IF;

ix := IN;



(* revision history
hm	28. jun. 2008
	original version

*)

END_FUNCTION_BLOCK

// POUs/Engineering/measurements/FLOW_METER
FUNCTION_BLOCK FLOW_METER
VAR_INPUT
	VX : REAL;
	E : BOOL;
	RST : BOOL;
END_VAR
VAR_INPUT CONSTANT
	PULSE_MODE : BOOL;
	UPDATE_TIME : TIME := t#1s;
END_VAR
VAR_OUTPUT
	F : REAL;
END_VAR
VAR_IN_OUT
	X : REAL;
	Y : UDINT;
END_VAR
VAR
	tx, tl : TIME;
	int1 : INTEGRATE;
	init: BOOL;
	e_last : BOOL;
	tmp: INT;
	x_last : REAL;
	y_last : UDINT;
END_VAR

(*
version 1.0	23. jan. 2011
programmer 	hugo
tested by	oscat

Flow meter measures flow according to gated time or pulses.

*)

IF NOT init THEN	(* init on power up *)
	init := TRUE;
	tl := tx;
	x_last := X;
	y_last := Y;
	int1.K := 2.7777777777777777E-4;
END_IF;

(* run integrator *)
int1(E := NOT (RST OR PULSE_MODE) AND E, X := VX, Y := X);	(* gated operation *)

IF RST THEN		(* reset *)
	X := 0.0;
	Y := 0;
	tl := tx;
	x_last := 0.0;
	y_last := 0;
ELSIF E AND PULSE_MODE THEN	(* check for pulse mode *)
	IF NOT e_last THEN X := X + VX; END_IF;
END_IF;
e_last := E;

(* reduce X to be less than 1 and increase Y respectively *)
IF X > 1.0 THEN
	tmp := FLOOR(X);
	Y := Y + INT_TO_UDINT(tmp);
	X := X - INT_TO_REAL(tmp);
END_IF;

(* calculate the current flow *)
tx := DWORD_TO_TIME(T_PLC_MS());
IF tx - tl >= UPDATE_TIME AND UPDATE_TIME > t#0s THEN
	F := (UDINT_TO_REAL(Y - y_last) + X - x_last) / TIME_TO_REAL(tx - tl) * 3.6E6;
	y_last := Y;
	x_last := X;
	tl := tx;
END_IF;



(* revision history
hm	23. jan. 2011	rev 1.0
	original version

*)

END_FUNCTION_BLOCK

// POUs/String/FSTRING_TO_BYTE
FUNCTION FSTRING_TO_BYTE : BYTE
VAR_INPUT
	IN : STRING(12);
END_VAR


(*
version 1.1	20. sep. 2008
programmer 	hugo
tested by		oscat

FSTRING_TO_BYTE converts a formatted string into a byte.
the string can be of the form 2#01010, 8#7234, 16#2AD3 and 1234

*)

IF LEFT(IN, 2) = '2#' THEN
	(* we need to convert binary *)
	FSTRING_TO_BYTE := BIN_TO_BYTE(RIGHT(in, LEN(in) - 2));
ELSIF LEFT(in, 2) = '8#' THEN
	(* weneed to convert octals *)
	FSTRING_TO_BYTE := OCT_TO_BYTE(RIGHT(in, LEN(in) - 2));
ELSIF LEFT(in, 3) = '16#' THEN
	(* we need to convert hexadecimal *)
	FSTRING_TO_BYTE := HEX_TO_BYTE(RIGHT(in, LEN(in) - 3));
ELSE
	(* we assume decimal representation *)
	FSTRING_TO_BYTE := DEC_TO_BYTE(CLEAN(in,'0123456789'));
END_IF;


(* revision histroy
hm	18. jun. 2008	rev 1.0
	original release

hm	20. sep. 2008	rev 1.1
	changed length of input string from 20 to 12
*)

END_FUNCTION

// POUs/String/OCT_TO_BYTE
FUNCTION OCT_TO_BYTE : BYTE
VAR_INPUT
	OCT : STRING(10);
END_VAR
VAR
	pt : POINTER TO BYTE;
	i: INT;
	X: BYTE;
	stop: INT;
END_VAR

(*
version 1.1	20. sep. 2008
programmer 	hugo
tested by		oscat

OCT_TO_BYTE converts a octagonal string into a byte.

*)

pt := ADR(oct);
stop := LEN(oct);
FOR I := 1 TO stop DO
	(* read the first character and subtract 48 to get value in decimal 0 = 48 *)
	x := pt^;
	(* calculate the value of the digit *)
	IF X > 47 AND x < 56 THEN
		OCT_TO_BYTE := SHL(OCT_TO_BYTE,3) + X - 48;
	END_IF;
	pt := pt + 1;
END_FOR;



(* revision histroy
hm	18. jun. 2008	rev 1.0
	original release

hm	20. sep. 2008	rev 1.1
	changed length of input string from 20 to 10

*)

END_FUNCTION

